BEGIN
   ZykIdx := 31;
   AntrMeld_chg_Idx := 0;
   Imp_Sek_Init := FALSE;
   OP_Mgr.Bed_aktiv := FALSE;
   OP_Mgr.Bed_ID := 0;
   OP_Mgr.Bed_Perm := 0;
   OP_Mgr.CtrlJob_act := FALSE;
   OP_Mgr.PicNum_AntrSub := FALSE;
   OP_Mgr.FM_PicNum_AntrSub := FALSE;
   OP_Mgr.PicNum_PrmSub_Rfrs := FALSE;
   OP_Mgr.PicNum_AntrSub_Rfrs := FALSE;
   OP_Mgr.MsgQuit_Zyk := FALSE;
   OP_Mgr.Bed_Perm_last := 0;
   OP_Mgr.Tmr_CtrlJob_MaxTime.ST := T#0MS;
   OP_Mgr.Tmr_CtrlJob_MaxTime.PT := T#0MS;
   OP_Mgr.Tmr_CtrlJob_MaxTime.RU := FALSE;
   OP_Mgr.Tmr_CtrlJob_MaxTime.IN := FALSE;
   OP_Mgr.Tmr_CtrlJob_BrkTime.ST := T#0MS;
   OP_Mgr.Tmr_CtrlJob_BrkTime.PT := T#0MS;
   OP_Mgr.Tmr_CtrlJob_BrkTime.RU := FALSE;
   OP_Mgr.Tmr_CtrlJob_BrkTime.IN := FALSE;
   OP_Mgr.Tmr_MsgQuit_Zyk.ST := T#0MS;
   OP_Mgr.Tmr_MsgQuit_Zyk.PT := T#0MS;
   OP_Mgr.Tmr_MsgQuit_Zyk.RU := FALSE;
   OP_Mgr.Tmr_MsgQuit_Zyk.IN := FALSE;
   OP_Mgr.CtrlJob_PicReq := 0;
   OP_Mgr.CtrlJob_PermReq := 0;
   OP_Mgr.OP_UserChg := 0;
   OP_Mgr.Antr_Idx_last := 0;
   OP_Mgr.AntrListChk_Idx := 113;
   OP_Mgr.SW_Hand_last := 0.0;
   BB_G1.Typ := 0;
   BB_G1.Idx := 0;
   BB_G1.BA_VW_Hand := FALSE;
   BB_G1.Tmr_VZ_Anlauf_Q := FALSE;
   BB_G1.SS := FALSE;
   BB_G1.SSnq := FALSE;
   BB_G1.SSfq := TRUE;
   BB_G1.nBB := FALSE;
   BB_G1.VW_Hand_St1 := FALSE;
   BB_G1.VW_Hand_St2 := FALSE;
   BB_G1.VW_Hand_Stop := FALSE;
   BB_G1.VW_Auto_St1 := FALSE;
   BB_G1.VW_Auto_St2 := FALSE;
   BB_G1.Anst_Req_St1 := FALSE;
   BB_G1.Anst_Req_St2 := FALSE;
   BB_G1.FM_Betrieb_Ein := FALSE;
   BB_G1.FM_Betrieb_Aus := TRUE;
   BB_G1.NLZ_MAZ_St1 := FALSE;
   BB_G1.NLZ_MAZ_St2 := FALSE;
   BB_G1.NLZ_Rev_SS_St1 := FALSE;
   BB_G1.NLZ_Rev_SS_St2 := FALSE;
   BB_G1.Th_St := FALSE;
   BB_G1.DMA_St := FALSE;
   BB_G1.DMZ_St := FALSE;
   BB_G1.FU_St := FALSE;
   BB_G1.TL_St := FALSE;
   BB_G1.UDr_St := FALSE;
   BB_G1.UeDr_St := FALSE;
   BB_G1.UT_St := FALSE;
   BB_G1.Le_St := FALSE;
   BB_G1.UeLM_St := FALSE;
   BB_G1.UeLE_St := FALSE;
   BB_G1.Kom_DP_St := FALSE;
   BB_G1.Kom_int_St := FALSE;
   BB_G1.int_St := FALSE;
   BB_G1.LZ_St := FALSE;
   BB_G1.BefLZ_St := FALSE;
   BB_G1.FM_GlobalQuit := FALSE;
   BB_G1.Quit_RST := FALSE;
   BB_G1.Tmr_VZ_Anlauf := 0;
   BB_G1.Tmr_VZ_ESZ := 0;
   BB_G1.Tmr_Th_St := 0;
   BB_G1.Tmr_DMA_St := 0;
   BB_G1.Tmr_DMZ_St := 0;
   BB_G1.Tmr_FU_St := 0;
   BB_G1.Tmr_TL_St := 0;
   BB_G1.Tmr_UDr_St := 0;
   BB_G1.Tmr_UeDr_St := 0;
   BB_G1.Tmr_UT_St := 0;
   BB_G1.Tmr_Le_St := 0;
   BB_G1.Tmr_UeLM_St := 0;
   BB_G1.Tmr_UeLE_St := 0;
   BB_G1.Tmr_Kom_DP_St := 0;
   BB_G1.Tmr_Kom_int_St := 0;
   BB_G1.Tmr_int_St := 0;
   BB_G1.Tmr_LZ_St := 0;
   BB_G1.Tmr_BefLZ_St := 0;
   BB_G1.Tmr_ASZ_St1 := 0;
   BB_G1.Tmr_ASZ_St2 := 0;
   BB_G1.Tmr_Rev_St1 := 0;
   BB_G1.Tmr_Rev_St2 := 0;
   BB_G1.BZ_ges_s := 507;
   BB_G1.Tmr_Quit_RST := 0;
   BB_G1.BEF_NHV.Bef.Bed_Res := FALSE;
   BB_G1.BEF_NHV.Bef.Bed_UV := FALSE;
   BB_G1.BEF_NHV.Bef.Bed_NHV := FALSE;
   BB_G1.BEF_NHV.Bef.Bed_PLS := FALSE;
   BB_G1.BEF_NHV.Bef.BA_Hand := FALSE;
   BB_G1.BEF_NHV.Bef.BA_Auto := FALSE;
   BB_G1.BEF_NHV.Bef.BF_Ein1 := FALSE;
   BB_G1.BEF_NHV.Bef.BF_Ein2 := FALSE;
   BB_G1.BEF_NHV.Bef.BF_Aus := FALSE;
   BB_G1.BEF_NHV.Bef.BZ_Res := FALSE;
   BB_G1.BEF_NHV.Bef.Res_10 := FALSE;
   BB_G1.BEF_NHV.Bef.Res_11 := FALSE;
   BB_G1.BEF_NHV.Bef.Res_12 := FALSE;
   BB_G1.BEF_NHV.Bef.Res_13 := FALSE;
   BB_G1.BEF_NHV.Bef.Res_14 := FALSE;
   BB_G1.BEF_NHV.Bef.Res_15 := FALSE;
   BB_G1.BEF_NHV.Bef.Res_16 := FALSE;
   BB_G1.BEF_NHV.Bef.Res_17 := FALSE;
   BB_G1.BEF_NHV.Bef.Res_18 := FALSE;
   BB_G1.BEF_NHV.Bef.Res_19 := FALSE;
   BB_G1.BEF_NHV.Bef.Res_20 := FALSE;
   BB_G1.BEF_NHV.Bef.Res_21 := FALSE;
   BB_G1.BEF_NHV.Bef.Res_22 := FALSE;
   BB_G1.BEF_NHV.Bef.Res_23 := FALSE;
   BB_G1.BEF_NHV.Bef.Res_24 := FALSE;
   BB_G1.BEF_NHV.Bef.Res_25 := FALSE;
   BB_G1.BEF_NHV.Bef.Res_26 := FALSE;
   BB_G1.BEF_NHV.Bef.Res_27 := FALSE;
   BB_G1.BEF_NHV.Bef.Res_28 := FALSE;
   BB_G1.BEF_NHV.Bef.Res_29 := FALSE;
   BB_G1.BEF_NHV.Bef.BF_Set_SW_chg := FALSE;
   BB_G1.BEF_NHV.Bef.BF_Quit := FALSE;
   BB_G1.BEF_NHV.SW_Hand := 0.0;
   BB_G2.Typ := 0;
   BB_G2.Idx := 1;
   BB_G2.BA_VW_Hand := FALSE;
   BB_G2.Tmr_VZ_Anlauf_Q := FALSE;
   BB_G2.SS := FALSE;
   BB_G2.SSnq := FALSE;
   BB_G2.SSfq := TRUE;
   BB_G2.nBB := FALSE;
   BB_G2.VW_Hand_St1 := FALSE;
   BB_G2.VW_Hand_St2 := FALSE;
   BB_G2.VW_Hand_Stop := FALSE;
   BB_G2.VW_Auto_St1 := FALSE;
   BB_G2.VW_Auto_St2 := FALSE;
   BB_G2.Anst_Req_St1 := FALSE;
   BB_G2.Anst_Req_St2 := FALSE;
   BB_G2.FM_Betrieb_Ein := FALSE;
   BB_G2.FM_Betrieb_Aus := TRUE;
   BB_G2.NLZ_MAZ_St1 := FALSE;
   BB_G2.NLZ_MAZ_St2 := FALSE;
   BB_G2.NLZ_Rev_SS_St1 := FALSE;
   BB_G2.NLZ_Rev_SS_St2 := FALSE;
   BB_G2.Th_St := FALSE;
   BB_G2.DMA_St := FALSE;
   BB_G2.DMZ_St := FALSE;
   BB_G2.FU_St := FALSE;
   BB_G2.TL_St := FALSE;
   BB_G2.UDr_St := FALSE;
   BB_G2.UeDr_St := FALSE;
   BB_G2.UT_St := FALSE;
   BB_G2.Le_St := FALSE;
   BB_G2.UeLM_St := FALSE;
   BB_G2.UeLE_St := FALSE;
   BB_G2.Kom_DP_St := FALSE;
   BB_G2.Kom_int_St := FALSE;
   BB_G2.int_St := FALSE;
   BB_G2.LZ_St := FALSE;
   BB_G2.BefLZ_St := FALSE;
   BB_G2.FM_GlobalQuit := FALSE;
   BB_G2.Quit_RST := FALSE;
   BB_G2.Tmr_VZ_Anlauf := 0;
   BB_G2.Tmr_VZ_ESZ := 0;
   BB_G2.Tmr_Th_St := 0;
   BB_G2.Tmr_DMA_St := 0;
   BB_G2.Tmr_DMZ_St := 0;
   BB_G2.Tmr_FU_St := 0;
   BB_G2.Tmr_TL_St := 0;
   BB_G2.Tmr_UDr_St := 0;
   BB_G2.Tmr_UeDr_St := 0;
   BB_G2.Tmr_UT_St := 0;
   BB_G2.Tmr_Le_St := 0;
   BB_G2.Tmr_UeLM_St := 0;
   BB_G2.Tmr_UeLE_St := 0;
   BB_G2.Tmr_Kom_DP_St := 0;
   BB_G2.Tmr_Kom_int_St := 0;
   BB_G2.Tmr_int_St := 0;
   BB_G2.Tmr_LZ_St := 0;
   BB_G2.Tmr_BefLZ_St := 0;
   BB_G2.Tmr_ASZ_St1 := 0;
   BB_G2.Tmr_ASZ_St2 := 0;
   BB_G2.Tmr_Rev_St1 := 0;
   BB_G2.Tmr_Rev_St2 := 0;
   BB_G2.BZ_ges_s := 3009;
   BB_G2.Tmr_Quit_RST := 0;
   BB_G2.BEF_NHV.Bef.Bed_Res := FALSE;
   BB_G2.BEF_NHV.Bef.Bed_UV := FALSE;
   BB_G2.BEF_NHV.Bef.Bed_NHV := FALSE;
   BB_G2.BEF_NHV.Bef.Bed_PLS := FALSE;
   BB_G2.BEF_NHV.Bef.BA_Hand := FALSE;
   BB_G2.BEF_NHV.Bef.BA_Auto := FALSE;
   BB_G2.BEF_NHV.Bef.BF_Ein1 := FALSE;
   BB_G2.BEF_NHV.Bef.BF_Ein2 := FALSE;
   BB_G2.BEF_NHV.Bef.BF_Aus := FALSE;
   BB_G2.BEF_NHV.Bef.BZ_Res := FALSE;
   BB_G2.BEF_NHV.Bef.Res_10 := FALSE;
   BB_G2.BEF_NHV.Bef.Res_11 := FALSE;
   BB_G2.BEF_NHV.Bef.Res_12 := FALSE;
   BB_G2.BEF_NHV.Bef.Res_13 := FALSE;
   BB_G2.BEF_NHV.Bef.Res_14 := FALSE;
   BB_G2.BEF_NHV.Bef.Res_15 := FALSE;
   BB_G2.BEF_NHV.Bef.Res_16 := FALSE;
   BB_G2.BEF_NHV.Bef.Res_17 := FALSE;
   BB_G2.BEF_NHV.Bef.Res_18 := FALSE;
   BB_G2.BEF_NHV.Bef.Res_19 := FALSE;
   BB_G2.BEF_NHV.Bef.Res_20 := FALSE;
   BB_G2.BEF_NHV.Bef.Res_21 := FALSE;
   BB_G2.BEF_NHV.Bef.Res_22 := FALSE;
   BB_G2.BEF_NHV.Bef.Res_23 := FALSE;
   BB_G2.BEF_NHV.Bef.Res_24 := FALSE;
   BB_G2.BEF_NHV.Bef.Res_25 := FALSE;
   BB_G2.BEF_NHV.Bef.Res_26 := FALSE;
   BB_G2.BEF_NHV.Bef.Res_27 := FALSE;
   BB_G2.BEF_NHV.Bef.Res_28 := FALSE;
   BB_G2.BEF_NHV.Bef.Res_29 := FALSE;
   BB_G2.BEF_NHV.Bef.BF_Set_SW_chg := FALSE;
   BB_G2.BEF_NHV.Bef.BF_Quit := FALSE;
   BB_G2.BEF_NHV.SW_Hand := 0.0;
   BB_G3.Typ := 0;
   BB_G3.Idx := 2;
   BB_G3.BA_VW_Hand := FALSE;
   BB_G3.Tmr_VZ_Anlauf_Q := FALSE;
   BB_G3.SS := FALSE;
   BB_G3.SSnq := FALSE;
   BB_G3.SSfq := TRUE;
   BB_G3.nBB := FALSE;
   BB_G3.VW_Hand_St1 := FALSE;
   BB_G3.VW_Hand_St2 := FALSE;
   BB_G3.VW_Hand_Stop := FALSE;
   BB_G3.VW_Auto_St1 := FALSE;
   BB_G3.VW_Auto_St2 := FALSE;
   BB_G3.Anst_Req_St1 := FALSE;
   BB_G3.Anst_Req_St2 := FALSE;
   BB_G3.FM_Betrieb_Ein := FALSE;
   BB_G3.FM_Betrieb_Aus := TRUE;
   BB_G3.NLZ_MAZ_St1 := FALSE;
   BB_G3.NLZ_MAZ_St2 := FALSE;
   BB_G3.NLZ_Rev_SS_St1 := FALSE;
   BB_G3.NLZ_Rev_SS_St2 := FALSE;
   BB_G3.Th_St := FALSE;
   BB_G3.DMA_St := FALSE;
   BB_G3.DMZ_St := FALSE;
   BB_G3.FU_St := FALSE;
   BB_G3.TL_St := FALSE;
   BB_G3.UDr_St := FALSE;
   BB_G3.UeDr_St := FALSE;
   BB_G3.UT_St := FALSE;
   BB_G3.Le_St := FALSE;
   BB_G3.UeLM_St := FALSE;
   BB_G3.UeLE_St := FALSE;
   BB_G3.Kom_DP_St := FALSE;
   BB_G3.Kom_int_St := FALSE;
   BB_G3.int_St := FALSE;
   BB_G3.LZ_St := FALSE;
   BB_G3.BefLZ_St := FALSE;
   BB_G3.FM_GlobalQuit := FALSE;
   BB_G3.Quit_RST := FALSE;
   BB_G3.Tmr_VZ_Anlauf := 0;
   BB_G3.Tmr_VZ_ESZ := 0;
   BB_G3.Tmr_Th_St := 0;
   BB_G3.Tmr_DMA_St := 0;
   BB_G3.Tmr_DMZ_St := 0;
   BB_G3.Tmr_FU_St := 0;
   BB_G3.Tmr_TL_St := 0;
   BB_G3.Tmr_UDr_St := 0;
   BB_G3.Tmr_UeDr_St := 0;
   BB_G3.Tmr_UT_St := 0;
   BB_G3.Tmr_Le_St := 0;
   BB_G3.Tmr_UeLM_St := 0;
   BB_G3.Tmr_UeLE_St := 0;
   BB_G3.Tmr_Kom_DP_St := 0;
   BB_G3.Tmr_Kom_int_St := 0;
   BB_G3.Tmr_int_St := 0;
   BB_G3.Tmr_LZ_St := 0;
   BB_G3.Tmr_BefLZ_St := 0;
   BB_G3.Tmr_ASZ_St1 := 0;
   BB_G3.Tmr_ASZ_St2 := 0;
   BB_G3.Tmr_Rev_St1 := 0;
   BB_G3.Tmr_Rev_St2 := 0;
   BB_G3.BZ_ges_s := 86;
   BB_G3.Tmr_Quit_RST := 0;
   BB_G3.BEF_NHV.Bef.Bed_Res := FALSE;
   BB_G3.BEF_NHV.Bef.Bed_UV := FALSE;
   BB_G3.BEF_NHV.Bef.Bed_NHV := FALSE;
   BB_G3.BEF_NHV.Bef.Bed_PLS := FALSE;
   BB_G3.BEF_NHV.Bef.BA_Hand := FALSE;
   BB_G3.BEF_NHV.Bef.BA_Auto := FALSE;
   BB_G3.BEF_NHV.Bef.BF_Ein1 := FALSE;
   BB_G3.BEF_NHV.Bef.BF_Ein2 := FALSE;
   BB_G3.BEF_NHV.Bef.BF_Aus := FALSE;
   BB_G3.BEF_NHV.Bef.BZ_Res := FALSE;
   BB_G3.BEF_NHV.Bef.Res_10 := FALSE;
   BB_G3.BEF_NHV.Bef.Res_11 := FALSE;
   BB_G3.BEF_NHV.Bef.Res_12 := FALSE;
   BB_G3.BEF_NHV.Bef.Res_13 := FALSE;
   BB_G3.BEF_NHV.Bef.Res_14 := FALSE;
   BB_G3.BEF_NHV.Bef.Res_15 := FALSE;
   BB_G3.BEF_NHV.Bef.Res_16 := FALSE;
   BB_G3.BEF_NHV.Bef.Res_17 := FALSE;
   BB_G3.BEF_NHV.Bef.Res_18 := FALSE;
   BB_G3.BEF_NHV.Bef.Res_19 := FALSE;
   BB_G3.BEF_NHV.Bef.Res_20 := FALSE;
   BB_G3.BEF_NHV.Bef.Res_21 := FALSE;
   BB_G3.BEF_NHV.Bef.Res_22 := FALSE;
   BB_G3.BEF_NHV.Bef.Res_23 := FALSE;
   BB_G3.BEF_NHV.Bef.Res_24 := FALSE;
   BB_G3.BEF_NHV.Bef.Res_25 := FALSE;
   BB_G3.BEF_NHV.Bef.Res_26 := FALSE;
   BB_G3.BEF_NHV.Bef.Res_27 := FALSE;
   BB_G3.BEF_NHV.Bef.Res_28 := FALSE;
   BB_G3.BEF_NHV.Bef.Res_29 := FALSE;
   BB_G3.BEF_NHV.Bef.BF_Set_SW_chg := FALSE;
   BB_G3.BEF_NHV.Bef.BF_Quit := FALSE;
   BB_G3.BEF_NHV.SW_Hand := 0.0;
   BB_SHL_G1.Typ := 0;
   BB_SHL_G1.Idx := 3;
   BB_SHL_G1.BA_VW_Hand := FALSE;
   BB_SHL_G1.Tmr_VZ_Anlauf_Q := FALSE;
   BB_SHL_G1.SS := FALSE;
   BB_SHL_G1.SSnq := FALSE;
   BB_SHL_G1.SSfq := TRUE;
   BB_SHL_G1.nBB := FALSE;
   BB_SHL_G1.VW_Hand_St1 := FALSE;
   BB_SHL_G1.VW_Hand_St2 := FALSE;
   BB_SHL_G1.VW_Hand_Stop := FALSE;
   BB_SHL_G1.VW_Auto_St1 := FALSE;
   BB_SHL_G1.VW_Auto_St2 := FALSE;
   BB_SHL_G1.Anst_Req_St1 := FALSE;
   BB_SHL_G1.Anst_Req_St2 := FALSE;
   BB_SHL_G1.FM_Betrieb_Ein := FALSE;
   BB_SHL_G1.FM_Betrieb_Aus := TRUE;
   BB_SHL_G1.NLZ_MAZ_St1 := FALSE;
   BB_SHL_G1.NLZ_MAZ_St2 := FALSE;
   BB_SHL_G1.NLZ_Rev_SS_St1 := FALSE;
   BB_SHL_G1.NLZ_Rev_SS_St2 := FALSE;
   BB_SHL_G1.Th_St := FALSE;
   BB_SHL_G1.DMA_St := FALSE;
   BB_SHL_G1.DMZ_St := FALSE;
   BB_SHL_G1.FU_St := FALSE;
   BB_SHL_G1.TL_St := FALSE;
   BB_SHL_G1.UDr_St := FALSE;
   BB_SHL_G1.UeDr_St := FALSE;
   BB_SHL_G1.UT_St := FALSE;
   BB_SHL_G1.Le_St := FALSE;
   BB_SHL_G1.UeLM_St := FALSE;
   BB_SHL_G1.UeLE_St := FALSE;
   BB_SHL_G1.Kom_DP_St := FALSE;
   BB_SHL_G1.Kom_int_St := FALSE;
   BB_SHL_G1.int_St := FALSE;
   BB_SHL_G1.LZ_St := FALSE;
   BB_SHL_G1.BefLZ_St := FALSE;
   BB_SHL_G1.FM_GlobalQuit := FALSE;
   BB_SHL_G1.Quit_RST := FALSE;
   BB_SHL_G1.Tmr_VZ_Anlauf := 0;
   BB_SHL_G1.Tmr_VZ_ESZ := 0;
   BB_SHL_G1.Tmr_Th_St := 0;
   BB_SHL_G1.Tmr_DMA_St := 0;
   BB_SHL_G1.Tmr_DMZ_St := 0;
   BB_SHL_G1.Tmr_FU_St := 0;
   BB_SHL_G1.Tmr_TL_St := 0;
   BB_SHL_G1.Tmr_UDr_St := 0;
   BB_SHL_G1.Tmr_UeDr_St := 0;
   BB_SHL_G1.Tmr_UT_St := 0;
   BB_SHL_G1.Tmr_Le_St := 0;
   BB_SHL_G1.Tmr_UeLM_St := 0;
   BB_SHL_G1.Tmr_UeLE_St := 0;
   BB_SHL_G1.Tmr_Kom_DP_St := 0;
   BB_SHL_G1.Tmr_Kom_int_St := 0;
   BB_SHL_G1.Tmr_int_St := 0;
   BB_SHL_G1.Tmr_LZ_St := 0;
   BB_SHL_G1.Tmr_BefLZ_St := 0;
   BB_SHL_G1.Tmr_ASZ_St1 := 0;
   BB_SHL_G1.Tmr_ASZ_St2 := 0;
   BB_SHL_G1.Tmr_Rev_St1 := 0;
   BB_SHL_G1.Tmr_Rev_St2 := 0;
   BB_SHL_G1.BZ_ges_s := 1574;
   BB_SHL_G1.Tmr_Quit_RST := 0;
   BB_SHL_G1.BEF_NHV.Bef.Bed_Res := FALSE;
   BB_SHL_G1.BEF_NHV.Bef.Bed_UV := FALSE;
   BB_SHL_G1.BEF_NHV.Bef.Bed_NHV := FALSE;
   BB_SHL_G1.BEF_NHV.Bef.Bed_PLS := FALSE;
   BB_SHL_G1.BEF_NHV.Bef.BA_Hand := FALSE;
   BB_SHL_G1.BEF_NHV.Bef.BA_Auto := FALSE;
   BB_SHL_G1.BEF_NHV.Bef.BF_Ein1 := FALSE;
   BB_SHL_G1.BEF_NHV.Bef.BF_Ein2 := FALSE;
   BB_SHL_G1.BEF_NHV.Bef.BF_Aus := FALSE;
   BB_SHL_G1.BEF_NHV.Bef.BZ_Res := FALSE;
   BB_SHL_G1.BEF_NHV.Bef.Res_10 := FALSE;
   BB_SHL_G1.BEF_NHV.Bef.Res_11 := FALSE;
   BB_SHL_G1.BEF_NHV.Bef.Res_12 := FALSE;
   BB_SHL_G1.BEF_NHV.Bef.Res_13 := FALSE;
   BB_SHL_G1.BEF_NHV.Bef.Res_14 := FALSE;
   BB_SHL_G1.BEF_NHV.Bef.Res_15 := FALSE;
   BB_SHL_G1.BEF_NHV.Bef.Res_16 := FALSE;
   BB_SHL_G1.BEF_NHV.Bef.Res_17 := FALSE;
   BB_SHL_G1.BEF_NHV.Bef.Res_18 := FALSE;
   BB_SHL_G1.BEF_NHV.Bef.Res_19 := FALSE;
   BB_SHL_G1.BEF_NHV.Bef.Res_20 := FALSE;
   BB_SHL_G1.BEF_NHV.Bef.Res_21 := FALSE;
   BB_SHL_G1.BEF_NHV.Bef.Res_22 := FALSE;
   BB_SHL_G1.BEF_NHV.Bef.Res_23 := FALSE;
   BB_SHL_G1.BEF_NHV.Bef.Res_24 := FALSE;
   BB_SHL_G1.BEF_NHV.Bef.Res_25 := FALSE;
   BB_SHL_G1.BEF_NHV.Bef.Res_26 := FALSE;
   BB_SHL_G1.BEF_NHV.Bef.Res_27 := FALSE;
   BB_SHL_G1.BEF_NHV.Bef.Res_28 := FALSE;
   BB_SHL_G1.BEF_NHV.Bef.Res_29 := FALSE;
   BB_SHL_G1.BEF_NHV.Bef.BF_Set_SW_chg := FALSE;
   BB_SHL_G1.BEF_NHV.Bef.BF_Quit := FALSE;
   BB_SHL_G1.BEF_NHV.SW_Hand := 0.0;
   BB_SHL_G2.Typ := 0;
   BB_SHL_G2.Idx := 4;
   BB_SHL_G2.BA_VW_Hand := FALSE;
   BB_SHL_G2.Tmr_VZ_Anlauf_Q := TRUE;
   BB_SHL_G2.SS := FALSE;
   BB_SHL_G2.SSnq := FALSE;
   BB_SHL_G2.SSfq := TRUE;
   BB_SHL_G2.nBB := FALSE;
   BB_SHL_G2.VW_Hand_St1 := FALSE;
   BB_SHL_G2.VW_Hand_St2 := FALSE;
   BB_SHL_G2.VW_Hand_Stop := FALSE;
   BB_SHL_G2.VW_Auto_St1 := FALSE;
   BB_SHL_G2.VW_Auto_St2 := FALSE;
   BB_SHL_G2.Anst_Req_St1 := FALSE;
   BB_SHL_G2.Anst_Req_St2 := FALSE;
   BB_SHL_G2.FM_Betrieb_Ein := TRUE;
   BB_SHL_G2.FM_Betrieb_Aus := FALSE;
   BB_SHL_G2.NLZ_MAZ_St1 := FALSE;
   BB_SHL_G2.NLZ_MAZ_St2 := FALSE;
   BB_SHL_G2.NLZ_Rev_SS_St1 := FALSE;
   BB_SHL_G2.NLZ_Rev_SS_St2 := FALSE;
   BB_SHL_G2.Th_St := FALSE;
   BB_SHL_G2.DMA_St := FALSE;
   BB_SHL_G2.DMZ_St := FALSE;
   BB_SHL_G2.FU_St := FALSE;
   BB_SHL_G2.TL_St := FALSE;
   BB_SHL_G2.UDr_St := FALSE;
   BB_SHL_G2.UeDr_St := FALSE;
   BB_SHL_G2.UT_St := FALSE;
   BB_SHL_G2.Le_St := FALSE;
   BB_SHL_G2.UeLM_St := FALSE;
   BB_SHL_G2.UeLE_St := FALSE;
   BB_SHL_G2.Kom_DP_St := FALSE;
   BB_SHL_G2.Kom_int_St := FALSE;
   BB_SHL_G2.int_St := FALSE;
   BB_SHL_G2.LZ_St := FALSE;
   BB_SHL_G2.BefLZ_St := FALSE;
   BB_SHL_G2.FM_GlobalQuit := FALSE;
   BB_SHL_G2.Quit_RST := FALSE;
   BB_SHL_G2.Tmr_VZ_Anlauf := 3;
   BB_SHL_G2.Tmr_VZ_ESZ := 0;
   BB_SHL_G2.Tmr_Th_St := 0;
   BB_SHL_G2.Tmr_DMA_St := 0;
   BB_SHL_G2.Tmr_DMZ_St := 0;
   BB_SHL_G2.Tmr_FU_St := 0;
   BB_SHL_G2.Tmr_TL_St := 0;
   BB_SHL_G2.Tmr_UDr_St := 0;
   BB_SHL_G2.Tmr_UeDr_St := 0;
   BB_SHL_G2.Tmr_UT_St := 0;
   BB_SHL_G2.Tmr_Le_St := 0;
   BB_SHL_G2.Tmr_UeLM_St := 0;
   BB_SHL_G2.Tmr_UeLE_St := 0;
   BB_SHL_G2.Tmr_Kom_DP_St := 0;
   BB_SHL_G2.Tmr_Kom_int_St := 0;
   BB_SHL_G2.Tmr_int_St := 0;
   BB_SHL_G2.Tmr_LZ_St := 0;
   BB_SHL_G2.Tmr_BefLZ_St := 0;
   BB_SHL_G2.Tmr_ASZ_St1 := 0;
   BB_SHL_G2.Tmr_ASZ_St2 := 0;
   BB_SHL_G2.Tmr_Rev_St1 := 0;
   BB_SHL_G2.Tmr_Rev_St2 := 0;
   BB_SHL_G2.BZ_ges_s := 4715;
   BB_SHL_G2.Tmr_Quit_RST := 0;
   BB_SHL_G2.BEF_NHV.Bef.Bed_Res := FALSE;
   BB_SHL_G2.BEF_NHV.Bef.Bed_UV := FALSE;
   BB_SHL_G2.BEF_NHV.Bef.Bed_NHV := FALSE;
   BB_SHL_G2.BEF_NHV.Bef.Bed_PLS := FALSE;
   BB_SHL_G2.BEF_NHV.Bef.BA_Hand := FALSE;
   BB_SHL_G2.BEF_NHV.Bef.BA_Auto := FALSE;
   BB_SHL_G2.BEF_NHV.Bef.BF_Ein1 := FALSE;
   BB_SHL_G2.BEF_NHV.Bef.BF_Ein2 := FALSE;
   BB_SHL_G2.BEF_NHV.Bef.BF_Aus := FALSE;
   BB_SHL_G2.BEF_NHV.Bef.BZ_Res := FALSE;
   BB_SHL_G2.BEF_NHV.Bef.Res_10 := FALSE;
   BB_SHL_G2.BEF_NHV.Bef.Res_11 := FALSE;
   BB_SHL_G2.BEF_NHV.Bef.Res_12 := FALSE;
   BB_SHL_G2.BEF_NHV.Bef.Res_13 := FALSE;
   BB_SHL_G2.BEF_NHV.Bef.Res_14 := FALSE;
   BB_SHL_G2.BEF_NHV.Bef.Res_15 := FALSE;
   BB_SHL_G2.BEF_NHV.Bef.Res_16 := FALSE;
   BB_SHL_G2.BEF_NHV.Bef.Res_17 := FALSE;
   BB_SHL_G2.BEF_NHV.Bef.Res_18 := FALSE;
   BB_SHL_G2.BEF_NHV.Bef.Res_19 := FALSE;
   BB_SHL_G2.BEF_NHV.Bef.Res_20 := FALSE;
   BB_SHL_G2.BEF_NHV.Bef.Res_21 := FALSE;
   BB_SHL_G2.BEF_NHV.Bef.Res_22 := FALSE;
   BB_SHL_G2.BEF_NHV.Bef.Res_23 := FALSE;
   BB_SHL_G2.BEF_NHV.Bef.Res_24 := FALSE;
   BB_SHL_G2.BEF_NHV.Bef.Res_25 := FALSE;
   BB_SHL_G2.BEF_NHV.Bef.Res_26 := FALSE;
   BB_SHL_G2.BEF_NHV.Bef.Res_27 := FALSE;
   BB_SHL_G2.BEF_NHV.Bef.Res_28 := FALSE;
   BB_SHL_G2.BEF_NHV.Bef.Res_29 := FALSE;
   BB_SHL_G2.BEF_NHV.Bef.BF_Set_SW_chg := FALSE;
   BB_SHL_G2.BEF_NHV.Bef.BF_Quit := FALSE;
   BB_SHL_G2.BEF_NHV.SW_Hand := 0.0;
   BB_SHL_G3.Typ := 0;
   BB_SHL_G3.Idx := 5;
   BB_SHL_G3.BA_VW_Hand := FALSE;
   BB_SHL_G3.Tmr_VZ_Anlauf_Q := FALSE;
   BB_SHL_G3.SS := FALSE;
   BB_SHL_G3.SSnq := FALSE;
   BB_SHL_G3.SSfq := TRUE;
   BB_SHL_G3.nBB := FALSE;
   BB_SHL_G3.VW_Hand_St1 := FALSE;
   BB_SHL_G3.VW_Hand_St2 := FALSE;
   BB_SHL_G3.VW_Hand_Stop := FALSE;
   BB_SHL_G3.VW_Auto_St1 := FALSE;
   BB_SHL_G3.VW_Auto_St2 := FALSE;
   BB_SHL_G3.Anst_Req_St1 := FALSE;
   BB_SHL_G3.Anst_Req_St2 := FALSE;
   BB_SHL_G3.FM_Betrieb_Ein := FALSE;
   BB_SHL_G3.FM_Betrieb_Aus := TRUE;
   BB_SHL_G3.NLZ_MAZ_St1 := FALSE;
   BB_SHL_G3.NLZ_MAZ_St2 := FALSE;
   BB_SHL_G3.NLZ_Rev_SS_St1 := FALSE;
   BB_SHL_G3.NLZ_Rev_SS_St2 := FALSE;
   BB_SHL_G3.Th_St := FALSE;
   BB_SHL_G3.DMA_St := FALSE;
   BB_SHL_G3.DMZ_St := FALSE;
   BB_SHL_G3.FU_St := FALSE;
   BB_SHL_G3.TL_St := FALSE;
   BB_SHL_G3.UDr_St := FALSE;
   BB_SHL_G3.UeDr_St := FALSE;
   BB_SHL_G3.UT_St := FALSE;
   BB_SHL_G3.Le_St := FALSE;
   BB_SHL_G3.UeLM_St := FALSE;
   BB_SHL_G3.UeLE_St := FALSE;
   BB_SHL_G3.Kom_DP_St := FALSE;
   BB_SHL_G3.Kom_int_St := FALSE;
   BB_SHL_G3.int_St := FALSE;
   BB_SHL_G3.LZ_St := FALSE;
   BB_SHL_G3.BefLZ_St := FALSE;
   BB_SHL_G3.FM_GlobalQuit := FALSE;
   BB_SHL_G3.Quit_RST := FALSE;
   BB_SHL_G3.Tmr_VZ_Anlauf := 0;
   BB_SHL_G3.Tmr_VZ_ESZ := 0;
   BB_SHL_G3.Tmr_Th_St := 0;
   BB_SHL_G3.Tmr_DMA_St := 0;
   BB_SHL_G3.Tmr_DMZ_St := 0;
   BB_SHL_G3.Tmr_FU_St := 0;
   BB_SHL_G3.Tmr_TL_St := 0;
   BB_SHL_G3.Tmr_UDr_St := 0;
   BB_SHL_G3.Tmr_UeDr_St := 0;
   BB_SHL_G3.Tmr_UT_St := 0;
   BB_SHL_G3.Tmr_Le_St := 0;
   BB_SHL_G3.Tmr_UeLM_St := 0;
   BB_SHL_G3.Tmr_UeLE_St := 0;
   BB_SHL_G3.Tmr_Kom_DP_St := 0;
   BB_SHL_G3.Tmr_Kom_int_St := 0;
   BB_SHL_G3.Tmr_int_St := 0;
   BB_SHL_G3.Tmr_LZ_St := 0;
   BB_SHL_G3.Tmr_BefLZ_St := 0;
   BB_SHL_G3.Tmr_ASZ_St1 := 0;
   BB_SHL_G3.Tmr_ASZ_St2 := 0;
   BB_SHL_G3.Tmr_Rev_St1 := 0;
   BB_SHL_G3.Tmr_Rev_St2 := 0;
   BB_SHL_G3.BZ_ges_s := 1375;
   BB_SHL_G3.Tmr_Quit_RST := 0;
   BB_SHL_G3.BEF_NHV.Bef.Bed_Res := FALSE;
   BB_SHL_G3.BEF_NHV.Bef.Bed_UV := FALSE;
   BB_SHL_G3.BEF_NHV.Bef.Bed_NHV := FALSE;
   BB_SHL_G3.BEF_NHV.Bef.Bed_PLS := FALSE;
   BB_SHL_G3.BEF_NHV.Bef.BA_Hand := FALSE;
   BB_SHL_G3.BEF_NHV.Bef.BA_Auto := FALSE;
   BB_SHL_G3.BEF_NHV.Bef.BF_Ein1 := FALSE;
   BB_SHL_G3.BEF_NHV.Bef.BF_Ein2 := FALSE;
   BB_SHL_G3.BEF_NHV.Bef.BF_Aus := FALSE;
   BB_SHL_G3.BEF_NHV.Bef.BZ_Res := FALSE;
   BB_SHL_G3.BEF_NHV.Bef.Res_10 := FALSE;
   BB_SHL_G3.BEF_NHV.Bef.Res_11 := FALSE;
   BB_SHL_G3.BEF_NHV.Bef.Res_12 := FALSE;
   BB_SHL_G3.BEF_NHV.Bef.Res_13 := FALSE;
   BB_SHL_G3.BEF_NHV.Bef.Res_14 := FALSE;
   BB_SHL_G3.BEF_NHV.Bef.Res_15 := FALSE;
   BB_SHL_G3.BEF_NHV.Bef.Res_16 := FALSE;
   BB_SHL_G3.BEF_NHV.Bef.Res_17 := FALSE;
   BB_SHL_G3.BEF_NHV.Bef.Res_18 := FALSE;
   BB_SHL_G3.BEF_NHV.Bef.Res_19 := FALSE;
   BB_SHL_G3.BEF_NHV.Bef.Res_20 := FALSE;
   BB_SHL_G3.BEF_NHV.Bef.Res_21 := FALSE;
   BB_SHL_G3.BEF_NHV.Bef.Res_22 := FALSE;
   BB_SHL_G3.BEF_NHV.Bef.Res_23 := FALSE;
   BB_SHL_G3.BEF_NHV.Bef.Res_24 := FALSE;
   BB_SHL_G3.BEF_NHV.Bef.Res_25 := FALSE;
   BB_SHL_G3.BEF_NHV.Bef.Res_26 := FALSE;
   BB_SHL_G3.BEF_NHV.Bef.Res_27 := FALSE;
   BB_SHL_G3.BEF_NHV.Bef.Res_28 := FALSE;
   BB_SHL_G3.BEF_NHV.Bef.Res_29 := FALSE;
   BB_SHL_G3.BEF_NHV.Bef.BF_Set_SW_chg := FALSE;
   BB_SHL_G3.BEF_NHV.Bef.BF_Quit := FALSE;
   BB_SHL_G3.BEF_NHV.SW_Hand := 0.0;
   BB_AV.Typ := 0;
   BB_AV.Idx := 6;
   BB_AV.BA_VW_Hand := FALSE;
   BB_AV.Tmr_VZ_Anlauf_Q := FALSE;
   BB_AV.SS := FALSE;
   BB_AV.SSnq := FALSE;
   BB_AV.SSfq := TRUE;
   BB_AV.nBB := FALSE;
   BB_AV.VW_Hand_St1 := FALSE;
   BB_AV.VW_Hand_St2 := FALSE;
   BB_AV.VW_Hand_Stop := FALSE;
   BB_AV.VW_Auto_St1 := FALSE;
   BB_AV.VW_Auto_St2 := FALSE;
   BB_AV.Anst_Req_St1 := FALSE;
   BB_AV.Anst_Req_St2 := FALSE;
   BB_AV.FM_Betrieb_Ein := FALSE;
   BB_AV.FM_Betrieb_Aus := TRUE;
   BB_AV.NLZ_MAZ_St1 := FALSE;
   BB_AV.NLZ_MAZ_St2 := FALSE;
   BB_AV.NLZ_Rev_SS_St1 := FALSE;
   BB_AV.NLZ_Rev_SS_St2 := FALSE;
   BB_AV.Th_St := FALSE;
   BB_AV.DMA_St := FALSE;
   BB_AV.DMZ_St := FALSE;
   BB_AV.FU_St := FALSE;
   BB_AV.TL_St := FALSE;
   BB_AV.UDr_St := FALSE;
   BB_AV.UeDr_St := FALSE;
   BB_AV.UT_St := FALSE;
   BB_AV.Le_St := FALSE;
   BB_AV.UeLM_St := FALSE;
   BB_AV.UeLE_St := FALSE;
   BB_AV.Kom_DP_St := FALSE;
   BB_AV.Kom_int_St := FALSE;
   BB_AV.int_St := FALSE;
   BB_AV.LZ_St := FALSE;
   BB_AV.BefLZ_St := FALSE;
   BB_AV.FM_GlobalQuit := FALSE;
   BB_AV.Quit_RST := FALSE;
   BB_AV.Tmr_VZ_Anlauf := 0;
   BB_AV.Tmr_VZ_ESZ := 0;
   BB_AV.Tmr_Th_St := 0;
   BB_AV.Tmr_DMA_St := 0;
   BB_AV.Tmr_DMZ_St := 0;
   BB_AV.Tmr_FU_St := 0;
   BB_AV.Tmr_TL_St := 0;
   BB_AV.Tmr_UDr_St := 0;
   BB_AV.Tmr_UeDr_St := 0;
   BB_AV.Tmr_UT_St := 0;
   BB_AV.Tmr_Le_St := 0;
   BB_AV.Tmr_UeLM_St := 0;
   BB_AV.Tmr_UeLE_St := 0;
   BB_AV.Tmr_Kom_DP_St := 0;
   BB_AV.Tmr_Kom_int_St := 0;
   BB_AV.Tmr_int_St := 0;
   BB_AV.Tmr_LZ_St := 0;
   BB_AV.Tmr_BefLZ_St := 0;
   BB_AV.Tmr_ASZ_St1 := 0;
   BB_AV.Tmr_ASZ_St2 := 0;
   BB_AV.Tmr_Rev_St1 := 0;
   BB_AV.Tmr_Rev_St2 := 0;
   BB_AV.BZ_ges_s := 0;
   BB_AV.Tmr_Quit_RST := 0;
   BB_AV.BEF_NHV.Bef.Bed_Res := FALSE;
   BB_AV.BEF_NHV.Bef.Bed_UV := FALSE;
   BB_AV.BEF_NHV.Bef.Bed_NHV := FALSE;
   BB_AV.BEF_NHV.Bef.Bed_PLS := FALSE;
   BB_AV.BEF_NHV.Bef.BA_Hand := FALSE;
   BB_AV.BEF_NHV.Bef.BA_Auto := FALSE;
   BB_AV.BEF_NHV.Bef.BF_Ein1 := FALSE;
   BB_AV.BEF_NHV.Bef.BF_Ein2 := FALSE;
   BB_AV.BEF_NHV.Bef.BF_Aus := FALSE;
   BB_AV.BEF_NHV.Bef.BZ_Res := FALSE;
   BB_AV.BEF_NHV.Bef.Res_10 := FALSE;
   BB_AV.BEF_NHV.Bef.Res_11 := FALSE;
   BB_AV.BEF_NHV.Bef.Res_12 := FALSE;
   BB_AV.BEF_NHV.Bef.Res_13 := FALSE;
   BB_AV.BEF_NHV.Bef.Res_14 := FALSE;
   BB_AV.BEF_NHV.Bef.Res_15 := FALSE;
   BB_AV.BEF_NHV.Bef.Res_16 := FALSE;
   BB_AV.BEF_NHV.Bef.Res_17 := FALSE;
   BB_AV.BEF_NHV.Bef.Res_18 := FALSE;
   BB_AV.BEF_NHV.Bef.Res_19 := FALSE;
   BB_AV.BEF_NHV.Bef.Res_20 := FALSE;
   BB_AV.BEF_NHV.Bef.Res_21 := FALSE;
   BB_AV.BEF_NHV.Bef.Res_22 := FALSE;
   BB_AV.BEF_NHV.Bef.Res_23 := FALSE;
   BB_AV.BEF_NHV.Bef.Res_24 := FALSE;
   BB_AV.BEF_NHV.Bef.Res_25 := FALSE;
   BB_AV.BEF_NHV.Bef.Res_26 := FALSE;
   BB_AV.BEF_NHV.Bef.Res_27 := FALSE;
   BB_AV.BEF_NHV.Bef.Res_28 := FALSE;
   BB_AV.BEF_NHV.Bef.Res_29 := FALSE;
   BB_AV.BEF_NHV.Bef.BF_Set_SW_chg := FALSE;
   BB_AV.BEF_NHV.Bef.BF_Quit := FALSE;
   BB_AV.BEF_NHV.SW_Hand := 0.0;
   BB_LS1.Typ := 5;
   BB_LS1.Idx := 7;
   BB_LS1.BA_VW_Hand := FALSE;
   BB_LS1.Tmr_VZ_Anlauf_Q := FALSE;
   BB_LS1.SS := FALSE;
   BB_LS1.SSnq := FALSE;
   BB_LS1.SSfq := TRUE;
   BB_LS1.nBB := FALSE;
   BB_LS1.VW_Hand_St1 := FALSE;
   BB_LS1.VW_Hand_St2 := FALSE;
   BB_LS1.VW_Hand_Stop := FALSE;
   BB_LS1.VW_Auto_St1 := FALSE;
   BB_LS1.VW_Auto_St2 := FALSE;
   BB_LS1.Anst_Req_St1 := FALSE;
   BB_LS1.Anst_Req_St2 := FALSE;
   BB_LS1.FM_Betrieb_Ein := FALSE;
   BB_LS1.FM_Betrieb_Aus := TRUE;
   BB_LS1.NLZ_MAZ_St1 := FALSE;
   BB_LS1.NLZ_MAZ_St2 := FALSE;
   BB_LS1.NLZ_Rev_SS_St1 := FALSE;
   BB_LS1.NLZ_Rev_SS_St2 := FALSE;
   BB_LS1.Th_St := FALSE;
   BB_LS1.DMA_St := FALSE;
   BB_LS1.DMZ_St := FALSE;
   BB_LS1.FU_St := FALSE;
   BB_LS1.TL_St := FALSE;
   BB_LS1.UDr_St := FALSE;
   BB_LS1.UeDr_St := FALSE;
   BB_LS1.UT_St := FALSE;
   BB_LS1.Le_St := FALSE;
   BB_LS1.UeLM_St := FALSE;
   BB_LS1.UeLE_St := FALSE;
   BB_LS1.Kom_DP_St := FALSE;
   BB_LS1.Kom_int_St := FALSE;
   BB_LS1.int_St := FALSE;
   BB_LS1.LZ_St := FALSE;
   BB_LS1.BefLZ_St := FALSE;
   BB_LS1.FM_GlobalQuit := FALSE;
   BB_LS1.Quit_RST := FALSE;
   BB_LS1.Tmr_VZ_Anlauf := 0;
   BB_LS1.Tmr_VZ_ESZ := 0;
   BB_LS1.Tmr_Th_St := 0;
   BB_LS1.Tmr_DMA_St := 0;
   BB_LS1.Tmr_DMZ_St := 0;
   BB_LS1.Tmr_FU_St := 0;
   BB_LS1.Tmr_TL_St := 0;
   BB_LS1.Tmr_UDr_St := 0;
   BB_LS1.Tmr_UeDr_St := 0;
   BB_LS1.Tmr_UT_St := 0;
   BB_LS1.Tmr_Le_St := 0;
   BB_LS1.Tmr_UeLM_St := 0;
   BB_LS1.Tmr_UeLE_St := 0;
   BB_LS1.Tmr_Kom_DP_St := 0;
   BB_LS1.Tmr_Kom_int_St := 0;
   BB_LS1.Tmr_int_St := 0;
   BB_LS1.Tmr_LZ_St := 0;
   BB_LS1.Tmr_BefLZ_St := 0;
   BB_LS1.Tmr_ASZ_St1 := 0;
   BB_LS1.Tmr_ASZ_St2 := 0;
   BB_LS1.Tmr_Rev_St1 := 0;
   BB_LS1.Tmr_Rev_St2 := 0;
   BB_LS1.BZ_ges_s := 127;
   BB_LS1.Tmr_Quit_RST := 0;
   BB_LS1.BEF_NHV.Bef.Bed_Res := FALSE;
   BB_LS1.BEF_NHV.Bef.Bed_UV := FALSE;
   BB_LS1.BEF_NHV.Bef.Bed_NHV := FALSE;
   BB_LS1.BEF_NHV.Bef.Bed_PLS := FALSE;
   BB_LS1.BEF_NHV.Bef.BA_Hand := FALSE;
   BB_LS1.BEF_NHV.Bef.BA_Auto := FALSE;
   BB_LS1.BEF_NHV.Bef.BF_Ein1 := FALSE;
   BB_LS1.BEF_NHV.Bef.BF_Ein2 := FALSE;
   BB_LS1.BEF_NHV.Bef.BF_Aus := FALSE;
   BB_LS1.BEF_NHV.Bef.BZ_Res := FALSE;
   BB_LS1.BEF_NHV.Bef.Res_10 := FALSE;
   BB_LS1.BEF_NHV.Bef.Res_11 := FALSE;
   BB_LS1.BEF_NHV.Bef.Res_12 := FALSE;
   BB_LS1.BEF_NHV.Bef.Res_13 := FALSE;
   BB_LS1.BEF_NHV.Bef.Res_14 := FALSE;
   BB_LS1.BEF_NHV.Bef.Res_15 := FALSE;
   BB_LS1.BEF_NHV.Bef.Res_16 := FALSE;
   BB_LS1.BEF_NHV.Bef.Res_17 := FALSE;
   BB_LS1.BEF_NHV.Bef.Res_18 := FALSE;
   BB_LS1.BEF_NHV.Bef.Res_19 := FALSE;
   BB_LS1.BEF_NHV.Bef.Res_20 := FALSE;
   BB_LS1.BEF_NHV.Bef.Res_21 := FALSE;
   BB_LS1.BEF_NHV.Bef.Res_22 := FALSE;
   BB_LS1.BEF_NHV.Bef.Res_23 := FALSE;
   BB_LS1.BEF_NHV.Bef.Res_24 := FALSE;
   BB_LS1.BEF_NHV.Bef.Res_25 := FALSE;
   BB_LS1.BEF_NHV.Bef.Res_26 := FALSE;
   BB_LS1.BEF_NHV.Bef.Res_27 := FALSE;
   BB_LS1.BEF_NHV.Bef.Res_28 := FALSE;
   BB_LS1.BEF_NHV.Bef.Res_29 := FALSE;
   BB_LS1.BEF_NHV.Bef.BF_Set_SW_chg := FALSE;
   BB_LS1.BEF_NHV.Bef.BF_Quit := FALSE;
   BB_LS1.BEF_NHV.SW_Hand := 0.0;
   BB_LS2.Typ := 5;
   BB_LS2.Idx := 8;
   BB_LS2.BA_VW_Hand := FALSE;
   BB_LS2.Tmr_VZ_Anlauf_Q := FALSE;
   BB_LS2.SS := FALSE;
   BB_LS2.SSnq := FALSE;
   BB_LS2.SSfq := TRUE;
   BB_LS2.nBB := FALSE;
   BB_LS2.VW_Hand_St1 := FALSE;
   BB_LS2.VW_Hand_St2 := FALSE;
   BB_LS2.VW_Hand_Stop := FALSE;
   BB_LS2.VW_Auto_St1 := FALSE;
   BB_LS2.VW_Auto_St2 := FALSE;
   BB_LS2.Anst_Req_St1 := FALSE;
   BB_LS2.Anst_Req_St2 := FALSE;
   BB_LS2.FM_Betrieb_Ein := FALSE;
   BB_LS2.FM_Betrieb_Aus := TRUE;
   BB_LS2.NLZ_MAZ_St1 := FALSE;
   BB_LS2.NLZ_MAZ_St2 := FALSE;
   BB_LS2.NLZ_Rev_SS_St1 := FALSE;
   BB_LS2.NLZ_Rev_SS_St2 := FALSE;
   BB_LS2.Th_St := FALSE;
   BB_LS2.DMA_St := FALSE;
   BB_LS2.DMZ_St := FALSE;
   BB_LS2.FU_St := FALSE;
   BB_LS2.TL_St := FALSE;
   BB_LS2.UDr_St := FALSE;
   BB_LS2.UeDr_St := FALSE;
   BB_LS2.UT_St := FALSE;
   BB_LS2.Le_St := FALSE;
   BB_LS2.UeLM_St := FALSE;
   BB_LS2.UeLE_St := FALSE;
   BB_LS2.Kom_DP_St := FALSE;
   BB_LS2.Kom_int_St := FALSE;
   BB_LS2.int_St := FALSE;
   BB_LS2.LZ_St := FALSE;
   BB_LS2.BefLZ_St := FALSE;
   BB_LS2.FM_GlobalQuit := FALSE;
   BB_LS2.Quit_RST := FALSE;
   BB_LS2.Tmr_VZ_Anlauf := 0;
   BB_LS2.Tmr_VZ_ESZ := 0;
   BB_LS2.Tmr_Th_St := 0;
   BB_LS2.Tmr_DMA_St := 0;
   BB_LS2.Tmr_DMZ_St := 0;
   BB_LS2.Tmr_FU_St := 0;
   BB_LS2.Tmr_TL_St := 0;
   BB_LS2.Tmr_UDr_St := 0;
   BB_LS2.Tmr_UeDr_St := 0;
   BB_LS2.Tmr_UT_St := 0;
   BB_LS2.Tmr_Le_St := 0;
   BB_LS2.Tmr_UeLM_St := 0;
   BB_LS2.Tmr_UeLE_St := 0;
   BB_LS2.Tmr_Kom_DP_St := 0;
   BB_LS2.Tmr_Kom_int_St := 0;
   BB_LS2.Tmr_int_St := 0;
   BB_LS2.Tmr_LZ_St := 0;
   BB_LS2.Tmr_BefLZ_St := 0;
   BB_LS2.Tmr_ASZ_St1 := 0;
   BB_LS2.Tmr_ASZ_St2 := 0;
   BB_LS2.Tmr_Rev_St1 := 0;
   BB_LS2.Tmr_Rev_St2 := 0;
   BB_LS2.BZ_ges_s := 298;
   BB_LS2.Tmr_Quit_RST := 0;
   BB_LS2.BEF_NHV.Bef.Bed_Res := FALSE;
   BB_LS2.BEF_NHV.Bef.Bed_UV := FALSE;
   BB_LS2.BEF_NHV.Bef.Bed_NHV := FALSE;
   BB_LS2.BEF_NHV.Bef.Bed_PLS := FALSE;
   BB_LS2.BEF_NHV.Bef.BA_Hand := FALSE;
   BB_LS2.BEF_NHV.Bef.BA_Auto := FALSE;
   BB_LS2.BEF_NHV.Bef.BF_Ein1 := FALSE;
   BB_LS2.BEF_NHV.Bef.BF_Ein2 := FALSE;
   BB_LS2.BEF_NHV.Bef.BF_Aus := FALSE;
   BB_LS2.BEF_NHV.Bef.BZ_Res := FALSE;
   BB_LS2.BEF_NHV.Bef.Res_10 := FALSE;
   BB_LS2.BEF_NHV.Bef.Res_11 := FALSE;
   BB_LS2.BEF_NHV.Bef.Res_12 := FALSE;
   BB_LS2.BEF_NHV.Bef.Res_13 := FALSE;
   BB_LS2.BEF_NHV.Bef.Res_14 := FALSE;
   BB_LS2.BEF_NHV.Bef.Res_15 := FALSE;
   BB_LS2.BEF_NHV.Bef.Res_16 := FALSE;
   BB_LS2.BEF_NHV.Bef.Res_17 := FALSE;
   BB_LS2.BEF_NHV.Bef.Res_18 := FALSE;
   BB_LS2.BEF_NHV.Bef.Res_19 := FALSE;
   BB_LS2.BEF_NHV.Bef.Res_20 := FALSE;
   BB_LS2.BEF_NHV.Bef.Res_21 := FALSE;
   BB_LS2.BEF_NHV.Bef.Res_22 := FALSE;
   BB_LS2.BEF_NHV.Bef.Res_23 := FALSE;
   BB_LS2.BEF_NHV.Bef.Res_24 := FALSE;
   BB_LS2.BEF_NHV.Bef.Res_25 := FALSE;
   BB_LS2.BEF_NHV.Bef.Res_26 := FALSE;
   BB_LS2.BEF_NHV.Bef.Res_27 := FALSE;
   BB_LS2.BEF_NHV.Bef.Res_28 := FALSE;
   BB_LS2.BEF_NHV.Bef.Res_29 := FALSE;
   BB_LS2.BEF_NHV.Bef.BF_Set_SW_chg := FALSE;
   BB_LS2.BEF_NHV.Bef.BF_Quit := FALSE;
   BB_LS2.BEF_NHV.SW_Hand := 0.0;
   BB1_RZP1.Typ := 0;
   BB1_RZP1.Idx := 9;
   BB1_RZP1.BA_VW_Hand := FALSE;
   BB1_RZP1.Tmr_VZ_Anlauf_Q := TRUE;
   BB1_RZP1.SS := FALSE;
   BB1_RZP1.SSnq := FALSE;
   BB1_RZP1.SSfq := TRUE;
   BB1_RZP1.nBB := FALSE;
   BB1_RZP1.VW_Hand_St1 := FALSE;
   BB1_RZP1.VW_Hand_St2 := FALSE;
   BB1_RZP1.VW_Hand_Stop := FALSE;
   BB1_RZP1.VW_Auto_St1 := TRUE;
   BB1_RZP1.VW_Auto_St2 := FALSE;
   BB1_RZP1.Anst_Req_St1 := TRUE;
   BB1_RZP1.Anst_Req_St2 := FALSE;
   BB1_RZP1.FM_Betrieb_Ein := TRUE;
   BB1_RZP1.FM_Betrieb_Aus := FALSE;
   BB1_RZP1.NLZ_MAZ_St1 := TRUE;
   BB1_RZP1.NLZ_MAZ_St2 := FALSE;
   BB1_RZP1.NLZ_Rev_SS_St1 := TRUE;
   BB1_RZP1.NLZ_Rev_SS_St2 := FALSE;
   BB1_RZP1.Th_St := FALSE;
   BB1_RZP1.DMA_St := FALSE;
   BB1_RZP1.DMZ_St := FALSE;
   BB1_RZP1.FU_St := FALSE;
   BB1_RZP1.TL_St := FALSE;
   BB1_RZP1.UDr_St := FALSE;
   BB1_RZP1.UeDr_St := FALSE;
   BB1_RZP1.UT_St := FALSE;
   BB1_RZP1.Le_St := FALSE;
   BB1_RZP1.UeLM_St := FALSE;
   BB1_RZP1.UeLE_St := FALSE;
   BB1_RZP1.Kom_DP_St := FALSE;
   BB1_RZP1.Kom_int_St := FALSE;
   BB1_RZP1.int_St := FALSE;
   BB1_RZP1.LZ_St := FALSE;
   BB1_RZP1.BefLZ_St := FALSE;
   BB1_RZP1.FM_GlobalQuit := FALSE;
   BB1_RZP1.Quit_RST := FALSE;
   BB1_RZP1.Tmr_VZ_Anlauf := 3;
   BB1_RZP1.Tmr_VZ_ESZ := 0;
   BB1_RZP1.Tmr_Th_St := 0;
   BB1_RZP1.Tmr_DMA_St := 0;
   BB1_RZP1.Tmr_DMZ_St := 0;
   BB1_RZP1.Tmr_FU_St := 0;
   BB1_RZP1.Tmr_TL_St := 0;
   BB1_RZP1.Tmr_UDr_St := 0;
   BB1_RZP1.Tmr_UeDr_St := 0;
   BB1_RZP1.Tmr_UT_St := 0;
   BB1_RZP1.Tmr_Le_St := 0;
   BB1_RZP1.Tmr_UeLM_St := 0;
   BB1_RZP1.Tmr_UeLE_St := 0;
   BB1_RZP1.Tmr_Kom_DP_St := 0;
   BB1_RZP1.Tmr_Kom_int_St := 0;
   BB1_RZP1.Tmr_int_St := 0;
   BB1_RZP1.Tmr_LZ_St := 0;
   BB1_RZP1.Tmr_BefLZ_St := 0;
   BB1_RZP1.Tmr_ASZ_St1 := 5;
   BB1_RZP1.Tmr_ASZ_St2 := 0;
   BB1_RZP1.Tmr_Rev_St1 := 10;
   BB1_RZP1.Tmr_Rev_St2 := 0;
   BB1_RZP1.BZ_ges_s := 2190;
   BB1_RZP1.Tmr_Quit_RST := 0;
   BB1_RZP1.BEF_NHV.Bef.Bed_Res := FALSE;
   BB1_RZP1.BEF_NHV.Bef.Bed_UV := FALSE;
   BB1_RZP1.BEF_NHV.Bef.Bed_NHV := FALSE;
   BB1_RZP1.BEF_NHV.Bef.Bed_PLS := FALSE;
   BB1_RZP1.BEF_NHV.Bef.BA_Hand := FALSE;
   BB1_RZP1.BEF_NHV.Bef.BA_Auto := FALSE;
   BB1_RZP1.BEF_NHV.Bef.BF_Ein1 := FALSE;
   BB1_RZP1.BEF_NHV.Bef.BF_Ein2 := FALSE;
   BB1_RZP1.BEF_NHV.Bef.BF_Aus := FALSE;
   BB1_RZP1.BEF_NHV.Bef.BZ_Res := FALSE;
   BB1_RZP1.BEF_NHV.Bef.Res_10 := FALSE;
   BB1_RZP1.BEF_NHV.Bef.Res_11 := FALSE;
   BB1_RZP1.BEF_NHV.Bef.Res_12 := FALSE;
   BB1_RZP1.BEF_NHV.Bef.Res_13 := FALSE;
   BB1_RZP1.BEF_NHV.Bef.Res_14 := FALSE;
   BB1_RZP1.BEF_NHV.Bef.Res_15 := FALSE;
   BB1_RZP1.BEF_NHV.Bef.Res_16 := FALSE;
   BB1_RZP1.BEF_NHV.Bef.Res_17 := FALSE;
   BB1_RZP1.BEF_NHV.Bef.Res_18 := FALSE;
   BB1_RZP1.BEF_NHV.Bef.Res_19 := FALSE;
   BB1_RZP1.BEF_NHV.Bef.Res_20 := FALSE;
   BB1_RZP1.BEF_NHV.Bef.Res_21 := FALSE;
   BB1_RZP1.BEF_NHV.Bef.Res_22 := FALSE;
   BB1_RZP1.BEF_NHV.Bef.Res_23 := FALSE;
   BB1_RZP1.BEF_NHV.Bef.Res_24 := FALSE;
   BB1_RZP1.BEF_NHV.Bef.Res_25 := FALSE;
   BB1_RZP1.BEF_NHV.Bef.Res_26 := FALSE;
   BB1_RZP1.BEF_NHV.Bef.Res_27 := FALSE;
   BB1_RZP1.BEF_NHV.Bef.Res_28 := FALSE;
   BB1_RZP1.BEF_NHV.Bef.Res_29 := FALSE;
   BB1_RZP1.BEF_NHV.Bef.BF_Set_SW_chg := FALSE;
   BB1_RZP1.BEF_NHV.Bef.BF_Quit := FALSE;
   BB1_RZP1.BEF_NHV.SW_Hand := 0.0;
   BB1_RZP2.Typ := 0;
   BB1_RZP2.Idx := 10;
   BB1_RZP2.BA_VW_Hand := FALSE;
   BB1_RZP2.Tmr_VZ_Anlauf_Q := FALSE;
   BB1_RZP2.SS := FALSE;
   BB1_RZP2.SSnq := FALSE;
   BB1_RZP2.SSfq := TRUE;
   BB1_RZP2.nBB := FALSE;
   BB1_RZP2.VW_Hand_St1 := FALSE;
   BB1_RZP2.VW_Hand_St2 := FALSE;
   BB1_RZP2.VW_Hand_Stop := FALSE;
   BB1_RZP2.VW_Auto_St1 := FALSE;
   BB1_RZP2.VW_Auto_St2 := FALSE;
   BB1_RZP2.Anst_Req_St1 := FALSE;
   BB1_RZP2.Anst_Req_St2 := FALSE;
   BB1_RZP2.FM_Betrieb_Ein := FALSE;
   BB1_RZP2.FM_Betrieb_Aus := TRUE;
   BB1_RZP2.NLZ_MAZ_St1 := FALSE;
   BB1_RZP2.NLZ_MAZ_St2 := FALSE;
   BB1_RZP2.NLZ_Rev_SS_St1 := FALSE;
   BB1_RZP2.NLZ_Rev_SS_St2 := FALSE;
   BB1_RZP2.Th_St := FALSE;
   BB1_RZP2.DMA_St := FALSE;
   BB1_RZP2.DMZ_St := FALSE;
   BB1_RZP2.FU_St := FALSE;
   BB1_RZP2.TL_St := FALSE;
   BB1_RZP2.UDr_St := FALSE;
   BB1_RZP2.UeDr_St := FALSE;
   BB1_RZP2.UT_St := FALSE;
   BB1_RZP2.Le_St := FALSE;
   BB1_RZP2.UeLM_St := FALSE;
   BB1_RZP2.UeLE_St := FALSE;
   BB1_RZP2.Kom_DP_St := FALSE;
   BB1_RZP2.Kom_int_St := FALSE;
   BB1_RZP2.int_St := FALSE;
   BB1_RZP2.LZ_St := FALSE;
   BB1_RZP2.BefLZ_St := FALSE;
   BB1_RZP2.FM_GlobalQuit := FALSE;
   BB1_RZP2.Quit_RST := FALSE;
   BB1_RZP2.Tmr_VZ_Anlauf := 0;
   BB1_RZP2.Tmr_VZ_ESZ := 0;
   BB1_RZP2.Tmr_Th_St := 0;
   BB1_RZP2.Tmr_DMA_St := 0;
   BB1_RZP2.Tmr_DMZ_St := 0;
   BB1_RZP2.Tmr_FU_St := 0;
   BB1_RZP2.Tmr_TL_St := 0;
   BB1_RZP2.Tmr_UDr_St := 0;
   BB1_RZP2.Tmr_UeDr_St := 0;
   BB1_RZP2.Tmr_UT_St := 0;
   BB1_RZP2.Tmr_Le_St := 0;
   BB1_RZP2.Tmr_UeLM_St := 0;
   BB1_RZP2.Tmr_UeLE_St := 0;
   BB1_RZP2.Tmr_Kom_DP_St := 0;
   BB1_RZP2.Tmr_Kom_int_St := 0;
   BB1_RZP2.Tmr_int_St := 0;
   BB1_RZP2.Tmr_LZ_St := 0;
   BB1_RZP2.Tmr_BefLZ_St := 0;
   BB1_RZP2.Tmr_ASZ_St1 := 0;
   BB1_RZP2.Tmr_ASZ_St2 := 0;
   BB1_RZP2.Tmr_Rev_St1 := 0;
   BB1_RZP2.Tmr_Rev_St2 := 0;
   BB1_RZP2.BZ_ges_s := 2591;
   BB1_RZP2.Tmr_Quit_RST := 0;
   BB1_RZP2.BEF_NHV.Bef.Bed_Res := FALSE;
   BB1_RZP2.BEF_NHV.Bef.Bed_UV := FALSE;
   BB1_RZP2.BEF_NHV.Bef.Bed_NHV := FALSE;
   BB1_RZP2.BEF_NHV.Bef.Bed_PLS := FALSE;
   BB1_RZP2.BEF_NHV.Bef.BA_Hand := FALSE;
   BB1_RZP2.BEF_NHV.Bef.BA_Auto := FALSE;
   BB1_RZP2.BEF_NHV.Bef.BF_Ein1 := FALSE;
   BB1_RZP2.BEF_NHV.Bef.BF_Ein2 := FALSE;
   BB1_RZP2.BEF_NHV.Bef.BF_Aus := FALSE;
   BB1_RZP2.BEF_NHV.Bef.BZ_Res := FALSE;
   BB1_RZP2.BEF_NHV.Bef.Res_10 := FALSE;
   BB1_RZP2.BEF_NHV.Bef.Res_11 := FALSE;
   BB1_RZP2.BEF_NHV.Bef.Res_12 := FALSE;
   BB1_RZP2.BEF_NHV.Bef.Res_13 := FALSE;
   BB1_RZP2.BEF_NHV.Bef.Res_14 := FALSE;
   BB1_RZP2.BEF_NHV.Bef.Res_15 := FALSE;
   BB1_RZP2.BEF_NHV.Bef.Res_16 := FALSE;
   BB1_RZP2.BEF_NHV.Bef.Res_17 := FALSE;
   BB1_RZP2.BEF_NHV.Bef.Res_18 := FALSE;
   BB1_RZP2.BEF_NHV.Bef.Res_19 := FALSE;
   BB1_RZP2.BEF_NHV.Bef.Res_20 := FALSE;
   BB1_RZP2.BEF_NHV.Bef.Res_21 := FALSE;
   BB1_RZP2.BEF_NHV.Bef.Res_22 := FALSE;
   BB1_RZP2.BEF_NHV.Bef.Res_23 := FALSE;
   BB1_RZP2.BEF_NHV.Bef.Res_24 := FALSE;
   BB1_RZP2.BEF_NHV.Bef.Res_25 := FALSE;
   BB1_RZP2.BEF_NHV.Bef.Res_26 := FALSE;
   BB1_RZP2.BEF_NHV.Bef.Res_27 := FALSE;
   BB1_RZP2.BEF_NHV.Bef.Res_28 := FALSE;
   BB1_RZP2.BEF_NHV.Bef.Res_29 := FALSE;
   BB1_RZP2.BEF_NHV.Bef.BF_Set_SW_chg := FALSE;
   BB1_RZP2.BEF_NHV.Bef.BF_Quit := FALSE;
   BB1_RZP2.BEF_NHV.SW_Hand := 0.0;
   BB1_UeSP.Typ := 0;
   BB1_UeSP.Idx := 11;
   BB1_UeSP.BA_VW_Hand := FALSE;
   BB1_UeSP.Tmr_VZ_Anlauf_Q := FALSE;
   BB1_UeSP.SS := FALSE;
   BB1_UeSP.SSnq := FALSE;
   BB1_UeSP.SSfq := TRUE;
   BB1_UeSP.nBB := FALSE;
   BB1_UeSP.VW_Hand_St1 := FALSE;
   BB1_UeSP.VW_Hand_St2 := FALSE;
   BB1_UeSP.VW_Hand_Stop := FALSE;
   BB1_UeSP.VW_Auto_St1 := FALSE;
   BB1_UeSP.VW_Auto_St2 := FALSE;
   BB1_UeSP.Anst_Req_St1 := FALSE;
   BB1_UeSP.Anst_Req_St2 := FALSE;
   BB1_UeSP.FM_Betrieb_Ein := FALSE;
   BB1_UeSP.FM_Betrieb_Aus := TRUE;
   BB1_UeSP.NLZ_MAZ_St1 := FALSE;
   BB1_UeSP.NLZ_MAZ_St2 := FALSE;
   BB1_UeSP.NLZ_Rev_SS_St1 := FALSE;
   BB1_UeSP.NLZ_Rev_SS_St2 := FALSE;
   BB1_UeSP.Th_St := FALSE;
   BB1_UeSP.DMA_St := FALSE;
   BB1_UeSP.DMZ_St := FALSE;
   BB1_UeSP.FU_St := FALSE;
   BB1_UeSP.TL_St := FALSE;
   BB1_UeSP.UDr_St := FALSE;
   BB1_UeSP.UeDr_St := FALSE;
   BB1_UeSP.UT_St := FALSE;
   BB1_UeSP.Le_St := FALSE;
   BB1_UeSP.UeLM_St := FALSE;
   BB1_UeSP.UeLE_St := FALSE;
   BB1_UeSP.Kom_DP_St := FALSE;
   BB1_UeSP.Kom_int_St := FALSE;
   BB1_UeSP.int_St := FALSE;
   BB1_UeSP.LZ_St := FALSE;
   BB1_UeSP.BefLZ_St := FALSE;
   BB1_UeSP.FM_GlobalQuit := FALSE;
   BB1_UeSP.Quit_RST := FALSE;
   BB1_UeSP.Tmr_VZ_Anlauf := 0;
   BB1_UeSP.Tmr_VZ_ESZ := 0;
   BB1_UeSP.Tmr_Th_St := 0;
   BB1_UeSP.Tmr_DMA_St := 0;
   BB1_UeSP.Tmr_DMZ_St := 0;
   BB1_UeSP.Tmr_FU_St := 0;
   BB1_UeSP.Tmr_TL_St := 0;
   BB1_UeSP.Tmr_UDr_St := 0;
   BB1_UeSP.Tmr_UeDr_St := 0;
   BB1_UeSP.Tmr_UT_St := 0;
   BB1_UeSP.Tmr_Le_St := 0;
   BB1_UeSP.Tmr_UeLM_St := 0;
   BB1_UeSP.Tmr_UeLE_St := 0;
   BB1_UeSP.Tmr_Kom_DP_St := 0;
   BB1_UeSP.Tmr_Kom_int_St := 0;
   BB1_UeSP.Tmr_int_St := 0;
   BB1_UeSP.Tmr_LZ_St := 0;
   BB1_UeSP.Tmr_BefLZ_St := 0;
   BB1_UeSP.Tmr_ASZ_St1 := 0;
   BB1_UeSP.Tmr_ASZ_St2 := 0;
   BB1_UeSP.Tmr_Rev_St1 := 0;
   BB1_UeSP.Tmr_Rev_St2 := 0;
   BB1_UeSP.BZ_ges_s := 2740;
   BB1_UeSP.Tmr_Quit_RST := 0;
   BB1_UeSP.BEF_NHV.Bef.Bed_Res := FALSE;
   BB1_UeSP.BEF_NHV.Bef.Bed_UV := FALSE;
   BB1_UeSP.BEF_NHV.Bef.Bed_NHV := FALSE;
   BB1_UeSP.BEF_NHV.Bef.Bed_PLS := FALSE;
   BB1_UeSP.BEF_NHV.Bef.BA_Hand := FALSE;
   BB1_UeSP.BEF_NHV.Bef.BA_Auto := FALSE;
   BB1_UeSP.BEF_NHV.Bef.BF_Ein1 := FALSE;
   BB1_UeSP.BEF_NHV.Bef.BF_Ein2 := FALSE;
   BB1_UeSP.BEF_NHV.Bef.BF_Aus := FALSE;
   BB1_UeSP.BEF_NHV.Bef.BZ_Res := FALSE;
   BB1_UeSP.BEF_NHV.Bef.Res_10 := FALSE;
   BB1_UeSP.BEF_NHV.Bef.Res_11 := FALSE;
   BB1_UeSP.BEF_NHV.Bef.Res_12 := FALSE;
   BB1_UeSP.BEF_NHV.Bef.Res_13 := FALSE;
   BB1_UeSP.BEF_NHV.Bef.Res_14 := FALSE;
   BB1_UeSP.BEF_NHV.Bef.Res_15 := FALSE;
   BB1_UeSP.BEF_NHV.Bef.Res_16 := FALSE;
   BB1_UeSP.BEF_NHV.Bef.Res_17 := FALSE;
   BB1_UeSP.BEF_NHV.Bef.Res_18 := FALSE;
   BB1_UeSP.BEF_NHV.Bef.Res_19 := FALSE;
   BB1_UeSP.BEF_NHV.Bef.Res_20 := FALSE;
   BB1_UeSP.BEF_NHV.Bef.Res_21 := FALSE;
   BB1_UeSP.BEF_NHV.Bef.Res_22 := FALSE;
   BB1_UeSP.BEF_NHV.Bef.Res_23 := FALSE;
   BB1_UeSP.BEF_NHV.Bef.Res_24 := FALSE;
   BB1_UeSP.BEF_NHV.Bef.Res_25 := FALSE;
   BB1_UeSP.BEF_NHV.Bef.Res_26 := FALSE;
   BB1_UeSP.BEF_NHV.Bef.Res_27 := FALSE;
   BB1_UeSP.BEF_NHV.Bef.Res_28 := FALSE;
   BB1_UeSP.BEF_NHV.Bef.Res_29 := FALSE;
   BB1_UeSP.BEF_NHV.Bef.BF_Set_SW_chg := FALSE;
   BB1_UeSP.BEF_NHV.Bef.BF_Quit := FALSE;
   BB1_UeSP.BEF_NHV.SW_Hand := 0.0;
   BB1_AS1.Typ := 5;
   BB1_AS1.Idx := 12;
   BB1_AS1.BA_VW_Hand := FALSE;
   BB1_AS1.Tmr_VZ_Anlauf_Q := FALSE;
   BB1_AS1.SS := FALSE;
   BB1_AS1.SSnq := FALSE;
   BB1_AS1.SSfq := TRUE;
   BB1_AS1.nBB := FALSE;
   BB1_AS1.VW_Hand_St1 := FALSE;
   BB1_AS1.VW_Hand_St2 := FALSE;
   BB1_AS1.VW_Hand_Stop := FALSE;
   BB1_AS1.VW_Auto_St1 := FALSE;
   BB1_AS1.VW_Auto_St2 := FALSE;
   BB1_AS1.Anst_Req_St1 := FALSE;
   BB1_AS1.Anst_Req_St2 := FALSE;
   BB1_AS1.FM_Betrieb_Ein := FALSE;
   BB1_AS1.FM_Betrieb_Aus := TRUE;
   BB1_AS1.NLZ_MAZ_St1 := FALSE;
   BB1_AS1.NLZ_MAZ_St2 := FALSE;
   BB1_AS1.NLZ_Rev_SS_St1 := FALSE;
   BB1_AS1.NLZ_Rev_SS_St2 := FALSE;
   BB1_AS1.Th_St := FALSE;
   BB1_AS1.DMA_St := FALSE;
   BB1_AS1.DMZ_St := FALSE;
   BB1_AS1.FU_St := FALSE;
   BB1_AS1.TL_St := FALSE;
   BB1_AS1.UDr_St := FALSE;
   BB1_AS1.UeDr_St := FALSE;
   BB1_AS1.UT_St := FALSE;
   BB1_AS1.Le_St := FALSE;
   BB1_AS1.UeLM_St := FALSE;
   BB1_AS1.UeLE_St := FALSE;
   BB1_AS1.Kom_DP_St := FALSE;
   BB1_AS1.Kom_int_St := FALSE;
   BB1_AS1.int_St := FALSE;
   BB1_AS1.LZ_St := FALSE;
   BB1_AS1.BefLZ_St := FALSE;
   BB1_AS1.FM_GlobalQuit := FALSE;
   BB1_AS1.Quit_RST := FALSE;
   BB1_AS1.Tmr_VZ_Anlauf := 0;
   BB1_AS1.Tmr_VZ_ESZ := 0;
   BB1_AS1.Tmr_Th_St := 0;
   BB1_AS1.Tmr_DMA_St := 0;
   BB1_AS1.Tmr_DMZ_St := 0;
   BB1_AS1.Tmr_FU_St := 0;
   BB1_AS1.Tmr_TL_St := 0;
   BB1_AS1.Tmr_UDr_St := 0;
   BB1_AS1.Tmr_UeDr_St := 0;
   BB1_AS1.Tmr_UT_St := 0;
   BB1_AS1.Tmr_Le_St := 0;
   BB1_AS1.Tmr_UeLM_St := 0;
   BB1_AS1.Tmr_UeLE_St := 0;
   BB1_AS1.Tmr_Kom_DP_St := 0;
   BB1_AS1.Tmr_Kom_int_St := 0;
   BB1_AS1.Tmr_int_St := 0;
   BB1_AS1.Tmr_LZ_St := 0;
   BB1_AS1.Tmr_BefLZ_St := 0;
   BB1_AS1.Tmr_ASZ_St1 := 0;
   BB1_AS1.Tmr_ASZ_St2 := 0;
   BB1_AS1.Tmr_Rev_St1 := 0;
   BB1_AS1.Tmr_Rev_St2 := 0;
   BB1_AS1.BZ_ges_s := 2050;
   BB1_AS1.Tmr_Quit_RST := 0;
   BB1_AS1.BEF_NHV.Bef.Bed_Res := FALSE;
   BB1_AS1.BEF_NHV.Bef.Bed_UV := FALSE;
   BB1_AS1.BEF_NHV.Bef.Bed_NHV := FALSE;
   BB1_AS1.BEF_NHV.Bef.Bed_PLS := FALSE;
   BB1_AS1.BEF_NHV.Bef.BA_Hand := FALSE;
   BB1_AS1.BEF_NHV.Bef.BA_Auto := FALSE;
   BB1_AS1.BEF_NHV.Bef.BF_Ein1 := FALSE;
   BB1_AS1.BEF_NHV.Bef.BF_Ein2 := FALSE;
   BB1_AS1.BEF_NHV.Bef.BF_Aus := FALSE;
   BB1_AS1.BEF_NHV.Bef.BZ_Res := FALSE;
   BB1_AS1.BEF_NHV.Bef.Res_10 := FALSE;
   BB1_AS1.BEF_NHV.Bef.Res_11 := FALSE;
   BB1_AS1.BEF_NHV.Bef.Res_12 := FALSE;
   BB1_AS1.BEF_NHV.Bef.Res_13 := FALSE;
   BB1_AS1.BEF_NHV.Bef.Res_14 := FALSE;
   BB1_AS1.BEF_NHV.Bef.Res_15 := FALSE;
   BB1_AS1.BEF_NHV.Bef.Res_16 := FALSE;
   BB1_AS1.BEF_NHV.Bef.Res_17 := FALSE;
   BB1_AS1.BEF_NHV.Bef.Res_18 := FALSE;
   BB1_AS1.BEF_NHV.Bef.Res_19 := FALSE;
   BB1_AS1.BEF_NHV.Bef.Res_20 := FALSE;
   BB1_AS1.BEF_NHV.Bef.Res_21 := FALSE;
   BB1_AS1.BEF_NHV.Bef.Res_22 := FALSE;
   BB1_AS1.BEF_NHV.Bef.Res_23 := FALSE;
   BB1_AS1.BEF_NHV.Bef.Res_24 := FALSE;
   BB1_AS1.BEF_NHV.Bef.Res_25 := FALSE;
   BB1_AS1.BEF_NHV.Bef.Res_26 := FALSE;
   BB1_AS1.BEF_NHV.Bef.Res_27 := FALSE;
   BB1_AS1.BEF_NHV.Bef.Res_28 := FALSE;
   BB1_AS1.BEF_NHV.Bef.Res_29 := FALSE;
   BB1_AS1.BEF_NHV.Bef.BF_Set_SW_chg := FALSE;
   BB1_AS1.BEF_NHV.Bef.BF_Quit := FALSE;
   BB1_AS1.BEF_NHV.SW_Hand := 0.0;
   BB1_AS2.Typ := 5;
   BB1_AS2.Idx := 13;
   BB1_AS2.BA_VW_Hand := FALSE;
   BB1_AS2.Tmr_VZ_Anlauf_Q := FALSE;
   BB1_AS2.SS := FALSE;
   BB1_AS2.SSnq := FALSE;
   BB1_AS2.SSfq := TRUE;
   BB1_AS2.nBB := FALSE;
   BB1_AS2.VW_Hand_St1 := FALSE;
   BB1_AS2.VW_Hand_St2 := FALSE;
   BB1_AS2.VW_Hand_Stop := FALSE;
   BB1_AS2.VW_Auto_St1 := FALSE;
   BB1_AS2.VW_Auto_St2 := FALSE;
   BB1_AS2.Anst_Req_St1 := FALSE;
   BB1_AS2.Anst_Req_St2 := FALSE;
   BB1_AS2.FM_Betrieb_Ein := FALSE;
   BB1_AS2.FM_Betrieb_Aus := TRUE;
   BB1_AS2.NLZ_MAZ_St1 := FALSE;
   BB1_AS2.NLZ_MAZ_St2 := FALSE;
   BB1_AS2.NLZ_Rev_SS_St1 := FALSE;
   BB1_AS2.NLZ_Rev_SS_St2 := FALSE;
   BB1_AS2.Th_St := FALSE;
   BB1_AS2.DMA_St := FALSE;
   BB1_AS2.DMZ_St := FALSE;
   BB1_AS2.FU_St := FALSE;
   BB1_AS2.TL_St := FALSE;
   BB1_AS2.UDr_St := FALSE;
   BB1_AS2.UeDr_St := FALSE;
   BB1_AS2.UT_St := FALSE;
   BB1_AS2.Le_St := FALSE;
   BB1_AS2.UeLM_St := FALSE;
   BB1_AS2.UeLE_St := FALSE;
   BB1_AS2.Kom_DP_St := FALSE;
   BB1_AS2.Kom_int_St := FALSE;
   BB1_AS2.int_St := FALSE;
   BB1_AS2.LZ_St := FALSE;
   BB1_AS2.BefLZ_St := FALSE;
   BB1_AS2.FM_GlobalQuit := FALSE;
   BB1_AS2.Quit_RST := FALSE;
   BB1_AS2.Tmr_VZ_Anlauf := 0;
   BB1_AS2.Tmr_VZ_ESZ := 0;
   BB1_AS2.Tmr_Th_St := 0;
   BB1_AS2.Tmr_DMA_St := 0;
   BB1_AS2.Tmr_DMZ_St := 0;
   BB1_AS2.Tmr_FU_St := 0;
   BB1_AS2.Tmr_TL_St := 0;
   BB1_AS2.Tmr_UDr_St := 0;
   BB1_AS2.Tmr_UeDr_St := 0;
   BB1_AS2.Tmr_UT_St := 0;
   BB1_AS2.Tmr_Le_St := 0;
   BB1_AS2.Tmr_UeLM_St := 0;
   BB1_AS2.Tmr_UeLE_St := 0;
   BB1_AS2.Tmr_Kom_DP_St := 0;
   BB1_AS2.Tmr_Kom_int_St := 0;
   BB1_AS2.Tmr_int_St := 0;
   BB1_AS2.Tmr_LZ_St := 0;
   BB1_AS2.Tmr_BefLZ_St := 0;
   BB1_AS2.Tmr_ASZ_St1 := 0;
   BB1_AS2.Tmr_ASZ_St2 := 0;
   BB1_AS2.Tmr_Rev_St1 := 0;
   BB1_AS2.Tmr_Rev_St2 := 0;
   BB1_AS2.BZ_ges_s := 1084;
   BB1_AS2.Tmr_Quit_RST := 0;
   BB1_AS2.BEF_NHV.Bef.Bed_Res := FALSE;
   BB1_AS2.BEF_NHV.Bef.Bed_UV := FALSE;
   BB1_AS2.BEF_NHV.Bef.Bed_NHV := FALSE;
   BB1_AS2.BEF_NHV.Bef.Bed_PLS := FALSE;
   BB1_AS2.BEF_NHV.Bef.BA_Hand := FALSE;
   BB1_AS2.BEF_NHV.Bef.BA_Auto := FALSE;
   BB1_AS2.BEF_NHV.Bef.BF_Ein1 := FALSE;
   BB1_AS2.BEF_NHV.Bef.BF_Ein2 := FALSE;
   BB1_AS2.BEF_NHV.Bef.BF_Aus := FALSE;
   BB1_AS2.BEF_NHV.Bef.BZ_Res := FALSE;
   BB1_AS2.BEF_NHV.Bef.Res_10 := FALSE;
   BB1_AS2.BEF_NHV.Bef.Res_11 := FALSE;
   BB1_AS2.BEF_NHV.Bef.Res_12 := FALSE;
   BB1_AS2.BEF_NHV.Bef.Res_13 := FALSE;
   BB1_AS2.BEF_NHV.Bef.Res_14 := FALSE;
   BB1_AS2.BEF_NHV.Bef.Res_15 := FALSE;
   BB1_AS2.BEF_NHV.Bef.Res_16 := FALSE;
   BB1_AS2.BEF_NHV.Bef.Res_17 := FALSE;
   BB1_AS2.BEF_NHV.Bef.Res_18 := FALSE;
   BB1_AS2.BEF_NHV.Bef.Res_19 := FALSE;
   BB1_AS2.BEF_NHV.Bef.Res_20 := FALSE;
   BB1_AS2.BEF_NHV.Bef.Res_21 := FALSE;
   BB1_AS2.BEF_NHV.Bef.Res_22 := FALSE;
   BB1_AS2.BEF_NHV.Bef.Res_23 := FALSE;
   BB1_AS2.BEF_NHV.Bef.Res_24 := FALSE;
   BB1_AS2.BEF_NHV.Bef.Res_25 := FALSE;
   BB1_AS2.BEF_NHV.Bef.Res_26 := FALSE;
   BB1_AS2.BEF_NHV.Bef.Res_27 := FALSE;
   BB1_AS2.BEF_NHV.Bef.Res_28 := FALSE;
   BB1_AS2.BEF_NHV.Bef.Res_29 := FALSE;
   BB1_AS2.BEF_NHV.Bef.BF_Set_SW_chg := FALSE;
   BB1_AS2.BEF_NHV.Bef.BF_Quit := FALSE;
   BB1_AS2.BEF_NHV.SW_Hand := 0.0;
   BB1_SR1.Typ := 7;
   BB1_SR1.Idx := 14;
   BB1_SR1.BA_VW_Hand := FALSE;
   BB1_SR1.Tmr_VZ_Anlauf_Q := FALSE;
   BB1_SR1.SS := FALSE;
   BB1_SR1.SSnq := FALSE;
   BB1_SR1.SSfq := TRUE;
   BB1_SR1.nBB := FALSE;
   BB1_SR1.VW_Hand_St1 := FALSE;
   BB1_SR1.VW_Hand_St2 := FALSE;
   BB1_SR1.VW_Hand_Stop := FALSE;
   BB1_SR1.VW_Auto_St1 := FALSE;
   BB1_SR1.VW_Auto_St2 := FALSE;
   BB1_SR1.Anst_Req_St1 := FALSE;
   BB1_SR1.Anst_Req_St2 := FALSE;
   BB1_SR1.FM_Betrieb_Ein := FALSE;
   BB1_SR1.FM_Betrieb_Aus := TRUE;
   BB1_SR1.NLZ_MAZ_St1 := FALSE;
   BB1_SR1.NLZ_MAZ_St2 := FALSE;
   BB1_SR1.NLZ_Rev_SS_St1 := FALSE;
   BB1_SR1.NLZ_Rev_SS_St2 := FALSE;
   BB1_SR1.Th_St := FALSE;
   BB1_SR1.DMA_St := FALSE;
   BB1_SR1.DMZ_St := FALSE;
   BB1_SR1.FU_St := FALSE;
   BB1_SR1.TL_St := FALSE;
   BB1_SR1.UDr_St := FALSE;
   BB1_SR1.UeDr_St := FALSE;
   BB1_SR1.UT_St := FALSE;
   BB1_SR1.Le_St := FALSE;
   BB1_SR1.UeLM_St := FALSE;
   BB1_SR1.UeLE_St := FALSE;
   BB1_SR1.Kom_DP_St := FALSE;
   BB1_SR1.Kom_int_St := FALSE;
   BB1_SR1.int_St := FALSE;
   BB1_SR1.LZ_St := FALSE;
   BB1_SR1.BefLZ_St := FALSE;
   BB1_SR1.FM_GlobalQuit := FALSE;
   BB1_SR1.Quit_RST := FALSE;
   BB1_SR1.Tmr_VZ_Anlauf := 0;
   BB1_SR1.Tmr_VZ_ESZ := 0;
   BB1_SR1.Tmr_Th_St := 0;
   BB1_SR1.Tmr_DMA_St := 0;
   BB1_SR1.Tmr_DMZ_St := 0;
   BB1_SR1.Tmr_FU_St := 0;
   BB1_SR1.Tmr_TL_St := 0;
   BB1_SR1.Tmr_UDr_St := 0;
   BB1_SR1.Tmr_UeDr_St := 0;
   BB1_SR1.Tmr_UT_St := 0;
   BB1_SR1.Tmr_Le_St := 0;
   BB1_SR1.Tmr_UeLM_St := 0;
   BB1_SR1.Tmr_UeLE_St := 0;
   BB1_SR1.Tmr_Kom_DP_St := 0;
   BB1_SR1.Tmr_Kom_int_St := 0;
   BB1_SR1.Tmr_int_St := 0;
   BB1_SR1.Tmr_LZ_St := 0;
   BB1_SR1.Tmr_BefLZ_St := 0;
   BB1_SR1.Tmr_ASZ_St1 := 0;
   BB1_SR1.Tmr_ASZ_St2 := 0;
   BB1_SR1.Tmr_Rev_St1 := 0;
   BB1_SR1.Tmr_Rev_St2 := 0;
   BB1_SR1.BZ_ges_s := 2705;
   BB1_SR1.Tmr_Quit_RST := 0;
   BB1_SR1.BEF_NHV.Bef.Bed_Res := FALSE;
   BB1_SR1.BEF_NHV.Bef.Bed_UV := FALSE;
   BB1_SR1.BEF_NHV.Bef.Bed_NHV := FALSE;
   BB1_SR1.BEF_NHV.Bef.Bed_PLS := FALSE;
   BB1_SR1.BEF_NHV.Bef.BA_Hand := FALSE;
   BB1_SR1.BEF_NHV.Bef.BA_Auto := FALSE;
   BB1_SR1.BEF_NHV.Bef.BF_Ein1 := FALSE;
   BB1_SR1.BEF_NHV.Bef.BF_Ein2 := FALSE;
   BB1_SR1.BEF_NHV.Bef.BF_Aus := FALSE;
   BB1_SR1.BEF_NHV.Bef.BZ_Res := FALSE;
   BB1_SR1.BEF_NHV.Bef.Res_10 := FALSE;
   BB1_SR1.BEF_NHV.Bef.Res_11 := FALSE;
   BB1_SR1.BEF_NHV.Bef.Res_12 := FALSE;
   BB1_SR1.BEF_NHV.Bef.Res_13 := FALSE;
   BB1_SR1.BEF_NHV.Bef.Res_14 := FALSE;
   BB1_SR1.BEF_NHV.Bef.Res_15 := FALSE;
   BB1_SR1.BEF_NHV.Bef.Res_16 := FALSE;
   BB1_SR1.BEF_NHV.Bef.Res_17 := FALSE;
   BB1_SR1.BEF_NHV.Bef.Res_18 := FALSE;
   BB1_SR1.BEF_NHV.Bef.Res_19 := FALSE;
   BB1_SR1.BEF_NHV.Bef.Res_20 := FALSE;
   BB1_SR1.BEF_NHV.Bef.Res_21 := FALSE;
   BB1_SR1.BEF_NHV.Bef.Res_22 := FALSE;
   BB1_SR1.BEF_NHV.Bef.Res_23 := FALSE;
   BB1_SR1.BEF_NHV.Bef.Res_24 := FALSE;
   BB1_SR1.BEF_NHV.Bef.Res_25 := FALSE;
   BB1_SR1.BEF_NHV.Bef.Res_26 := FALSE;
   BB1_SR1.BEF_NHV.Bef.Res_27 := FALSE;
   BB1_SR1.BEF_NHV.Bef.Res_28 := FALSE;
   BB1_SR1.BEF_NHV.Bef.Res_29 := FALSE;
   BB1_SR1.BEF_NHV.Bef.BF_Set_SW_chg := FALSE;
   BB1_SR1.BEF_NHV.Bef.BF_Quit := FALSE;
   BB1_SR1.BEF_NHV.SW_Hand := 0.0;
   BB1_SR2.Typ := 7;
   BB1_SR2.Idx := 15;
   BB1_SR2.BA_VW_Hand := FALSE;
   BB1_SR2.Tmr_VZ_Anlauf_Q := FALSE;
   BB1_SR2.SS := FALSE;
   BB1_SR2.SSnq := FALSE;
   BB1_SR2.SSfq := TRUE;
   BB1_SR2.nBB := FALSE;
   BB1_SR2.VW_Hand_St1 := FALSE;
   BB1_SR2.VW_Hand_St2 := FALSE;
   BB1_SR2.VW_Hand_Stop := FALSE;
   BB1_SR2.VW_Auto_St1 := FALSE;
   BB1_SR2.VW_Auto_St2 := FALSE;
   BB1_SR2.Anst_Req_St1 := FALSE;
   BB1_SR2.Anst_Req_St2 := FALSE;
   BB1_SR2.FM_Betrieb_Ein := FALSE;
   BB1_SR2.FM_Betrieb_Aus := TRUE;
   BB1_SR2.NLZ_MAZ_St1 := FALSE;
   BB1_SR2.NLZ_MAZ_St2 := FALSE;
   BB1_SR2.NLZ_Rev_SS_St1 := FALSE;
   BB1_SR2.NLZ_Rev_SS_St2 := FALSE;
   BB1_SR2.Th_St := FALSE;
   BB1_SR2.DMA_St := FALSE;
   BB1_SR2.DMZ_St := FALSE;
   BB1_SR2.FU_St := FALSE;
   BB1_SR2.TL_St := FALSE;
   BB1_SR2.UDr_St := FALSE;
   BB1_SR2.UeDr_St := FALSE;
   BB1_SR2.UT_St := FALSE;
   BB1_SR2.Le_St := FALSE;
   BB1_SR2.UeLM_St := FALSE;
   BB1_SR2.UeLE_St := FALSE;
   BB1_SR2.Kom_DP_St := FALSE;
   BB1_SR2.Kom_int_St := FALSE;
   BB1_SR2.int_St := FALSE;
   BB1_SR2.LZ_St := FALSE;
   BB1_SR2.BefLZ_St := FALSE;
   BB1_SR2.FM_GlobalQuit := FALSE;
   BB1_SR2.Quit_RST := FALSE;
   BB1_SR2.Tmr_VZ_Anlauf := 0;
   BB1_SR2.Tmr_VZ_ESZ := 0;
   BB1_SR2.Tmr_Th_St := 0;
   BB1_SR2.Tmr_DMA_St := 0;
   BB1_SR2.Tmr_DMZ_St := 0;
   BB1_SR2.Tmr_FU_St := 0;
   BB1_SR2.Tmr_TL_St := 0;
   BB1_SR2.Tmr_UDr_St := 0;
   BB1_SR2.Tmr_UeDr_St := 0;
   BB1_SR2.Tmr_UT_St := 0;
   BB1_SR2.Tmr_Le_St := 0;
   BB1_SR2.Tmr_UeLM_St := 0;
   BB1_SR2.Tmr_UeLE_St := 0;
   BB1_SR2.Tmr_Kom_DP_St := 0;
   BB1_SR2.Tmr_Kom_int_St := 0;
   BB1_SR2.Tmr_int_St := 0;
   BB1_SR2.Tmr_LZ_St := 0;
   BB1_SR2.Tmr_BefLZ_St := 0;
   BB1_SR2.Tmr_ASZ_St1 := 0;
   BB1_SR2.Tmr_ASZ_St2 := 0;
   BB1_SR2.Tmr_Rev_St1 := 0;
   BB1_SR2.Tmr_Rev_St2 := 0;
   BB1_SR2.BZ_ges_s := 2698;
   BB1_SR2.Tmr_Quit_RST := 0;
   BB1_SR2.BEF_NHV.Bef.Bed_Res := FALSE;
   BB1_SR2.BEF_NHV.Bef.Bed_UV := FALSE;
   BB1_SR2.BEF_NHV.Bef.Bed_NHV := FALSE;
   BB1_SR2.BEF_NHV.Bef.Bed_PLS := FALSE;
   BB1_SR2.BEF_NHV.Bef.BA_Hand := FALSE;
   BB1_SR2.BEF_NHV.Bef.BA_Auto := FALSE;
   BB1_SR2.BEF_NHV.Bef.BF_Ein1 := FALSE;
   BB1_SR2.BEF_NHV.Bef.BF_Ein2 := FALSE;
   BB1_SR2.BEF_NHV.Bef.BF_Aus := FALSE;
   BB1_SR2.BEF_NHV.Bef.BZ_Res := FALSE;
   BB1_SR2.BEF_NHV.Bef.Res_10 := FALSE;
   BB1_SR2.BEF_NHV.Bef.Res_11 := FALSE;
   BB1_SR2.BEF_NHV.Bef.Res_12 := FALSE;
   BB1_SR2.BEF_NHV.Bef.Res_13 := FALSE;
   BB1_SR2.BEF_NHV.Bef.Res_14 := FALSE;
   BB1_SR2.BEF_NHV.Bef.Res_15 := FALSE;
   BB1_SR2.BEF_NHV.Bef.Res_16 := FALSE;
   BB1_SR2.BEF_NHV.Bef.Res_17 := FALSE;
   BB1_SR2.BEF_NHV.Bef.Res_18 := FALSE;
   BB1_SR2.BEF_NHV.Bef.Res_19 := FALSE;
   BB1_SR2.BEF_NHV.Bef.Res_20 := FALSE;
   BB1_SR2.BEF_NHV.Bef.Res_21 := FALSE;
   BB1_SR2.BEF_NHV.Bef.Res_22 := FALSE;
   BB1_SR2.BEF_NHV.Bef.Res_23 := FALSE;
   BB1_SR2.BEF_NHV.Bef.Res_24 := FALSE;
   BB1_SR2.BEF_NHV.Bef.Res_25 := FALSE;
   BB1_SR2.BEF_NHV.Bef.Res_26 := FALSE;
   BB1_SR2.BEF_NHV.Bef.Res_27 := FALSE;
   BB1_SR2.BEF_NHV.Bef.Res_28 := FALSE;
   BB1_SR2.BEF_NHV.Bef.Res_29 := FALSE;
   BB1_SR2.BEF_NHV.Bef.BF_Set_SW_chg := FALSE;
   BB1_SR2.BEF_NHV.Bef.BF_Quit := FALSE;
   BB1_SR2.BEF_NHV.SW_Hand := 0.0;
   BB2_RZP1.Typ := 0;
   BB2_RZP1.Idx := 16;
   BB2_RZP1.BA_VW_Hand := FALSE;
   BB2_RZP1.Tmr_VZ_Anlauf_Q := FALSE;
   BB2_RZP1.SS := FALSE;
   BB2_RZP1.SSnq := FALSE;
   BB2_RZP1.SSfq := TRUE;
   BB2_RZP1.nBB := FALSE;
   BB2_RZP1.VW_Hand_St1 := FALSE;
   BB2_RZP1.VW_Hand_St2 := FALSE;
   BB2_RZP1.VW_Hand_Stop := FALSE;
   BB2_RZP1.VW_Auto_St1 := FALSE;
   BB2_RZP1.VW_Auto_St2 := FALSE;
   BB2_RZP1.Anst_Req_St1 := FALSE;
   BB2_RZP1.Anst_Req_St2 := FALSE;
   BB2_RZP1.FM_Betrieb_Ein := FALSE;
   BB2_RZP1.FM_Betrieb_Aus := TRUE;
   BB2_RZP1.NLZ_MAZ_St1 := FALSE;
   BB2_RZP1.NLZ_MAZ_St2 := FALSE;
   BB2_RZP1.NLZ_Rev_SS_St1 := FALSE;
   BB2_RZP1.NLZ_Rev_SS_St2 := FALSE;
   BB2_RZP1.Th_St := FALSE;
   BB2_RZP1.DMA_St := FALSE;
   BB2_RZP1.DMZ_St := FALSE;
   BB2_RZP1.FU_St := FALSE;
   BB2_RZP1.TL_St := FALSE;
   BB2_RZP1.UDr_St := FALSE;
   BB2_RZP1.UeDr_St := FALSE;
   BB2_RZP1.UT_St := FALSE;
   BB2_RZP1.Le_St := FALSE;
   BB2_RZP1.UeLM_St := FALSE;
   BB2_RZP1.UeLE_St := FALSE;
   BB2_RZP1.Kom_DP_St := FALSE;
   BB2_RZP1.Kom_int_St := FALSE;
   BB2_RZP1.int_St := FALSE;
   BB2_RZP1.LZ_St := FALSE;
   BB2_RZP1.BefLZ_St := FALSE;
   BB2_RZP1.FM_GlobalQuit := FALSE;
   BB2_RZP1.Quit_RST := FALSE;
   BB2_RZP1.Tmr_VZ_Anlauf := 0;
   BB2_RZP1.Tmr_VZ_ESZ := 0;
   BB2_RZP1.Tmr_Th_St := 0;
   BB2_RZP1.Tmr_DMA_St := 0;
   BB2_RZP1.Tmr_DMZ_St := 0;
   BB2_RZP1.Tmr_FU_St := 0;
   BB2_RZP1.Tmr_TL_St := 0;
   BB2_RZP1.Tmr_UDr_St := 0;
   BB2_RZP1.Tmr_UeDr_St := 0;
   BB2_RZP1.Tmr_UT_St := 0;
   BB2_RZP1.Tmr_Le_St := 0;
   BB2_RZP1.Tmr_UeLM_St := 0;
   BB2_RZP1.Tmr_UeLE_St := 0;
   BB2_RZP1.Tmr_Kom_DP_St := 0;
   BB2_RZP1.Tmr_Kom_int_St := 0;
   BB2_RZP1.Tmr_int_St := 0;
   BB2_RZP1.Tmr_LZ_St := 0;
   BB2_RZP1.Tmr_BefLZ_St := 0;
   BB2_RZP1.Tmr_ASZ_St1 := 0;
   BB2_RZP1.Tmr_ASZ_St2 := 0;
   BB2_RZP1.Tmr_Rev_St1 := 0;
   BB2_RZP1.Tmr_Rev_St2 := 0;
   BB2_RZP1.BZ_ges_s := 2197;
   BB2_RZP1.Tmr_Quit_RST := 0;
   BB2_RZP1.BEF_NHV.Bef.Bed_Res := FALSE;
   BB2_RZP1.BEF_NHV.Bef.Bed_UV := FALSE;
   BB2_RZP1.BEF_NHV.Bef.Bed_NHV := FALSE;
   BB2_RZP1.BEF_NHV.Bef.Bed_PLS := FALSE;
   BB2_RZP1.BEF_NHV.Bef.BA_Hand := FALSE;
   BB2_RZP1.BEF_NHV.Bef.BA_Auto := FALSE;
   BB2_RZP1.BEF_NHV.Bef.BF_Ein1 := FALSE;
   BB2_RZP1.BEF_NHV.Bef.BF_Ein2 := FALSE;
   BB2_RZP1.BEF_NHV.Bef.BF_Aus := FALSE;
   BB2_RZP1.BEF_NHV.Bef.BZ_Res := FALSE;
   BB2_RZP1.BEF_NHV.Bef.Res_10 := FALSE;
   BB2_RZP1.BEF_NHV.Bef.Res_11 := FALSE;
   BB2_RZP1.BEF_NHV.Bef.Res_12 := FALSE;
   BB2_RZP1.BEF_NHV.Bef.Res_13 := FALSE;
   BB2_RZP1.BEF_NHV.Bef.Res_14 := FALSE;
   BB2_RZP1.BEF_NHV.Bef.Res_15 := FALSE;
   BB2_RZP1.BEF_NHV.Bef.Res_16 := FALSE;
   BB2_RZP1.BEF_NHV.Bef.Res_17 := FALSE;
   BB2_RZP1.BEF_NHV.Bef.Res_18 := FALSE;
   BB2_RZP1.BEF_NHV.Bef.Res_19 := FALSE;
   BB2_RZP1.BEF_NHV.Bef.Res_20 := FALSE;
   BB2_RZP1.BEF_NHV.Bef.Res_21 := FALSE;
   BB2_RZP1.BEF_NHV.Bef.Res_22 := FALSE;
   BB2_RZP1.BEF_NHV.Bef.Res_23 := FALSE;
   BB2_RZP1.BEF_NHV.Bef.Res_24 := FALSE;
   BB2_RZP1.BEF_NHV.Bef.Res_25 := FALSE;
   BB2_RZP1.BEF_NHV.Bef.Res_26 := FALSE;
   BB2_RZP1.BEF_NHV.Bef.Res_27 := FALSE;
   BB2_RZP1.BEF_NHV.Bef.Res_28 := FALSE;
   BB2_RZP1.BEF_NHV.Bef.Res_29 := FALSE;
   BB2_RZP1.BEF_NHV.Bef.BF_Set_SW_chg := FALSE;
   BB2_RZP1.BEF_NHV.Bef.BF_Quit := FALSE;
   BB2_RZP1.BEF_NHV.SW_Hand := 0.0;
   BB2_RZP2.Typ := 0;
   BB2_RZP2.Idx := 17;
   BB2_RZP2.BA_VW_Hand := FALSE;
   BB2_RZP2.Tmr_VZ_Anlauf_Q := FALSE;
   BB2_RZP2.SS := FALSE;
   BB2_RZP2.SSnq := FALSE;
   BB2_RZP2.SSfq := TRUE;
   BB2_RZP2.nBB := FALSE;
   BB2_RZP2.VW_Hand_St1 := FALSE;
   BB2_RZP2.VW_Hand_St2 := FALSE;
   BB2_RZP2.VW_Hand_Stop := FALSE;
   BB2_RZP2.VW_Auto_St1 := FALSE;
   BB2_RZP2.VW_Auto_St2 := FALSE;
   BB2_RZP2.Anst_Req_St1 := FALSE;
   BB2_RZP2.Anst_Req_St2 := FALSE;
   BB2_RZP2.FM_Betrieb_Ein := FALSE;
   BB2_RZP2.FM_Betrieb_Aus := TRUE;
   BB2_RZP2.NLZ_MAZ_St1 := FALSE;
   BB2_RZP2.NLZ_MAZ_St2 := FALSE;
   BB2_RZP2.NLZ_Rev_SS_St1 := FALSE;
   BB2_RZP2.NLZ_Rev_SS_St2 := FALSE;
   BB2_RZP2.Th_St := FALSE;
   BB2_RZP2.DMA_St := FALSE;
   BB2_RZP2.DMZ_St := FALSE;
   BB2_RZP2.FU_St := FALSE;
   BB2_RZP2.TL_St := FALSE;
   BB2_RZP2.UDr_St := FALSE;
   BB2_RZP2.UeDr_St := FALSE;
   BB2_RZP2.UT_St := FALSE;
   BB2_RZP2.Le_St := FALSE;
   BB2_RZP2.UeLM_St := FALSE;
   BB2_RZP2.UeLE_St := FALSE;
   BB2_RZP2.Kom_DP_St := FALSE;
   BB2_RZP2.Kom_int_St := FALSE;
   BB2_RZP2.int_St := FALSE;
   BB2_RZP2.LZ_St := FALSE;
   BB2_RZP2.BefLZ_St := FALSE;
   BB2_RZP2.FM_GlobalQuit := FALSE;
   BB2_RZP2.Quit_RST := FALSE;
   BB2_RZP2.Tmr_VZ_Anlauf := 0;
   BB2_RZP2.Tmr_VZ_ESZ := 0;
   BB2_RZP2.Tmr_Th_St := 0;
   BB2_RZP2.Tmr_DMA_St := 0;
   BB2_RZP2.Tmr_DMZ_St := 0;
   BB2_RZP2.Tmr_FU_St := 0;
   BB2_RZP2.Tmr_TL_St := 0;
   BB2_RZP2.Tmr_UDr_St := 0;
   BB2_RZP2.Tmr_UeDr_St := 0;
   BB2_RZP2.Tmr_UT_St := 0;
   BB2_RZP2.Tmr_Le_St := 0;
   BB2_RZP2.Tmr_UeLM_St := 0;
   BB2_RZP2.Tmr_UeLE_St := 0;
   BB2_RZP2.Tmr_Kom_DP_St := 0;
   BB2_RZP2.Tmr_Kom_int_St := 0;
   BB2_RZP2.Tmr_int_St := 0;
   BB2_RZP2.Tmr_LZ_St := 0;
   BB2_RZP2.Tmr_BefLZ_St := 0;
   BB2_RZP2.Tmr_ASZ_St1 := 0;
   BB2_RZP2.Tmr_ASZ_St2 := 0;
   BB2_RZP2.Tmr_Rev_St1 := 0;
   BB2_RZP2.Tmr_Rev_St2 := 0;
   BB2_RZP2.BZ_ges_s := 2494;
   BB2_RZP2.Tmr_Quit_RST := 0;
   BB2_RZP2.BEF_NHV.Bef.Bed_Res := FALSE;
   BB2_RZP2.BEF_NHV.Bef.Bed_UV := FALSE;
   BB2_RZP2.BEF_NHV.Bef.Bed_NHV := FALSE;
   BB2_RZP2.BEF_NHV.Bef.Bed_PLS := FALSE;
   BB2_RZP2.BEF_NHV.Bef.BA_Hand := FALSE;
   BB2_RZP2.BEF_NHV.Bef.BA_Auto := FALSE;
   BB2_RZP2.BEF_NHV.Bef.BF_Ein1 := FALSE;
   BB2_RZP2.BEF_NHV.Bef.BF_Ein2 := FALSE;
   BB2_RZP2.BEF_NHV.Bef.BF_Aus := FALSE;
   BB2_RZP2.BEF_NHV.Bef.BZ_Res := FALSE;
   BB2_RZP2.BEF_NHV.Bef.Res_10 := FALSE;
   BB2_RZP2.BEF_NHV.Bef.Res_11 := FALSE;
   BB2_RZP2.BEF_NHV.Bef.Res_12 := FALSE;
   BB2_RZP2.BEF_NHV.Bef.Res_13 := FALSE;
   BB2_RZP2.BEF_NHV.Bef.Res_14 := FALSE;
   BB2_RZP2.BEF_NHV.Bef.Res_15 := FALSE;
   BB2_RZP2.BEF_NHV.Bef.Res_16 := FALSE;
   BB2_RZP2.BEF_NHV.Bef.Res_17 := FALSE;
   BB2_RZP2.BEF_NHV.Bef.Res_18 := FALSE;
   BB2_RZP2.BEF_NHV.Bef.Res_19 := FALSE;
   BB2_RZP2.BEF_NHV.Bef.Res_20 := FALSE;
   BB2_RZP2.BEF_NHV.Bef.Res_21 := FALSE;
   BB2_RZP2.BEF_NHV.Bef.Res_22 := FALSE;
   BB2_RZP2.BEF_NHV.Bef.Res_23 := FALSE;
   BB2_RZP2.BEF_NHV.Bef.Res_24 := FALSE;
   BB2_RZP2.BEF_NHV.Bef.Res_25 := FALSE;
   BB2_RZP2.BEF_NHV.Bef.Res_26 := FALSE;
   BB2_RZP2.BEF_NHV.Bef.Res_27 := FALSE;
   BB2_RZP2.BEF_NHV.Bef.Res_28 := FALSE;
   BB2_RZP2.BEF_NHV.Bef.Res_29 := FALSE;
   BB2_RZP2.BEF_NHV.Bef.BF_Set_SW_chg := FALSE;
   BB2_RZP2.BEF_NHV.Bef.BF_Quit := FALSE;
   BB2_RZP2.BEF_NHV.SW_Hand := 0.0;
   BB2_UeSP.Typ := 0;
   BB2_UeSP.Idx := 18;
   BB2_UeSP.BA_VW_Hand := FALSE;
   BB2_UeSP.Tmr_VZ_Anlauf_Q := FALSE;
   BB2_UeSP.SS := FALSE;
   BB2_UeSP.SSnq := FALSE;
   BB2_UeSP.SSfq := TRUE;
   BB2_UeSP.nBB := FALSE;
   BB2_UeSP.VW_Hand_St1 := FALSE;
   BB2_UeSP.VW_Hand_St2 := FALSE;
   BB2_UeSP.VW_Hand_Stop := FALSE;
   BB2_UeSP.VW_Auto_St1 := FALSE;
   BB2_UeSP.VW_Auto_St2 := FALSE;
   BB2_UeSP.Anst_Req_St1 := FALSE;
   BB2_UeSP.Anst_Req_St2 := FALSE;
   BB2_UeSP.FM_Betrieb_Ein := FALSE;
   BB2_UeSP.FM_Betrieb_Aus := TRUE;
   BB2_UeSP.NLZ_MAZ_St1 := FALSE;
   BB2_UeSP.NLZ_MAZ_St2 := FALSE;
   BB2_UeSP.NLZ_Rev_SS_St1 := FALSE;
   BB2_UeSP.NLZ_Rev_SS_St2 := FALSE;
   BB2_UeSP.Th_St := FALSE;
   BB2_UeSP.DMA_St := FALSE;
   BB2_UeSP.DMZ_St := FALSE;
   BB2_UeSP.FU_St := FALSE;
   BB2_UeSP.TL_St := FALSE;
   BB2_UeSP.UDr_St := FALSE;
   BB2_UeSP.UeDr_St := FALSE;
   BB2_UeSP.UT_St := FALSE;
   BB2_UeSP.Le_St := FALSE;
   BB2_UeSP.UeLM_St := FALSE;
   BB2_UeSP.UeLE_St := FALSE;
   BB2_UeSP.Kom_DP_St := FALSE;
   BB2_UeSP.Kom_int_St := FALSE;
   BB2_UeSP.int_St := FALSE;
   BB2_UeSP.LZ_St := FALSE;
   BB2_UeSP.BefLZ_St := FALSE;
   BB2_UeSP.FM_GlobalQuit := FALSE;
   BB2_UeSP.Quit_RST := FALSE;
   BB2_UeSP.Tmr_VZ_Anlauf := 0;
   BB2_UeSP.Tmr_VZ_ESZ := 0;
   BB2_UeSP.Tmr_Th_St := 0;
   BB2_UeSP.Tmr_DMA_St := 0;
   BB2_UeSP.Tmr_DMZ_St := 0;
   BB2_UeSP.Tmr_FU_St := 0;
   BB2_UeSP.Tmr_TL_St := 0;
   BB2_UeSP.Tmr_UDr_St := 0;
   BB2_UeSP.Tmr_UeDr_St := 0;
   BB2_UeSP.Tmr_UT_St := 0;
   BB2_UeSP.Tmr_Le_St := 0;
   BB2_UeSP.Tmr_UeLM_St := 0;
   BB2_UeSP.Tmr_UeLE_St := 0;
   BB2_UeSP.Tmr_Kom_DP_St := 0;
   BB2_UeSP.Tmr_Kom_int_St := 0;
   BB2_UeSP.Tmr_int_St := 0;
   BB2_UeSP.Tmr_LZ_St := 0;
   BB2_UeSP.Tmr_BefLZ_St := 0;
   BB2_UeSP.Tmr_ASZ_St1 := 0;
   BB2_UeSP.Tmr_ASZ_St2 := 0;
   BB2_UeSP.Tmr_Rev_St1 := 0;
   BB2_UeSP.Tmr_Rev_St2 := 0;
   BB2_UeSP.BZ_ges_s := 375;
   BB2_UeSP.Tmr_Quit_RST := 0;
   BB2_UeSP.BEF_NHV.Bef.Bed_Res := FALSE;
   BB2_UeSP.BEF_NHV.Bef.Bed_UV := FALSE;
   BB2_UeSP.BEF_NHV.Bef.Bed_NHV := FALSE;
   BB2_UeSP.BEF_NHV.Bef.Bed_PLS := FALSE;
   BB2_UeSP.BEF_NHV.Bef.BA_Hand := FALSE;
   BB2_UeSP.BEF_NHV.Bef.BA_Auto := FALSE;
   BB2_UeSP.BEF_NHV.Bef.BF_Ein1 := FALSE;
   BB2_UeSP.BEF_NHV.Bef.BF_Ein2 := FALSE;
   BB2_UeSP.BEF_NHV.Bef.BF_Aus := FALSE;
   BB2_UeSP.BEF_NHV.Bef.BZ_Res := FALSE;
   BB2_UeSP.BEF_NHV.Bef.Res_10 := FALSE;
   BB2_UeSP.BEF_NHV.Bef.Res_11 := FALSE;
   BB2_UeSP.BEF_NHV.Bef.Res_12 := FALSE;
   BB2_UeSP.BEF_NHV.Bef.Res_13 := FALSE;
   BB2_UeSP.BEF_NHV.Bef.Res_14 := FALSE;
   BB2_UeSP.BEF_NHV.Bef.Res_15 := FALSE;
   BB2_UeSP.BEF_NHV.Bef.Res_16 := FALSE;
   BB2_UeSP.BEF_NHV.Bef.Res_17 := FALSE;
   BB2_UeSP.BEF_NHV.Bef.Res_18 := FALSE;
   BB2_UeSP.BEF_NHV.Bef.Res_19 := FALSE;
   BB2_UeSP.BEF_NHV.Bef.Res_20 := FALSE;
   BB2_UeSP.BEF_NHV.Bef.Res_21 := FALSE;
   BB2_UeSP.BEF_NHV.Bef.Res_22 := FALSE;
   BB2_UeSP.BEF_NHV.Bef.Res_23 := FALSE;
   BB2_UeSP.BEF_NHV.Bef.Res_24 := FALSE;
   BB2_UeSP.BEF_NHV.Bef.Res_25 := FALSE;
   BB2_UeSP.BEF_NHV.Bef.Res_26 := FALSE;
   BB2_UeSP.BEF_NHV.Bef.Res_27 := FALSE;
   BB2_UeSP.BEF_NHV.Bef.Res_28 := FALSE;
   BB2_UeSP.BEF_NHV.Bef.Res_29 := FALSE;
   BB2_UeSP.BEF_NHV.Bef.BF_Set_SW_chg := FALSE;
   BB2_UeSP.BEF_NHV.Bef.BF_Quit := FALSE;
   BB2_UeSP.BEF_NHV.SW_Hand := 0.0;
   BB2_AS1.Typ := 5;
   BB2_AS1.Idx := 19;
   BB2_AS1.BA_VW_Hand := FALSE;
   BB2_AS1.Tmr_VZ_Anlauf_Q := FALSE;
   BB2_AS1.SS := FALSE;
   BB2_AS1.SSnq := FALSE;
   BB2_AS1.SSfq := TRUE;
   BB2_AS1.nBB := FALSE;
   BB2_AS1.VW_Hand_St1 := FALSE;
   BB2_AS1.VW_Hand_St2 := FALSE;
   BB2_AS1.VW_Hand_Stop := FALSE;
   BB2_AS1.VW_Auto_St1 := FALSE;
   BB2_AS1.VW_Auto_St2 := FALSE;
   BB2_AS1.Anst_Req_St1 := FALSE;
   BB2_AS1.Anst_Req_St2 := FALSE;
   BB2_AS1.FM_Betrieb_Ein := FALSE;
   BB2_AS1.FM_Betrieb_Aus := TRUE;
   BB2_AS1.NLZ_MAZ_St1 := FALSE;
   BB2_AS1.NLZ_MAZ_St2 := FALSE;
   BB2_AS1.NLZ_Rev_SS_St1 := FALSE;
   BB2_AS1.NLZ_Rev_SS_St2 := FALSE;
   BB2_AS1.Th_St := FALSE;
   BB2_AS1.DMA_St := FALSE;
   BB2_AS1.DMZ_St := FALSE;
   BB2_AS1.FU_St := FALSE;
   BB2_AS1.TL_St := FALSE;
   BB2_AS1.UDr_St := FALSE;
   BB2_AS1.UeDr_St := FALSE;
   BB2_AS1.UT_St := FALSE;
   BB2_AS1.Le_St := FALSE;
   BB2_AS1.UeLM_St := FALSE;
   BB2_AS1.UeLE_St := FALSE;
   BB2_AS1.Kom_DP_St := FALSE;
   BB2_AS1.Kom_int_St := FALSE;
   BB2_AS1.int_St := FALSE;
   BB2_AS1.LZ_St := FALSE;
   BB2_AS1.BefLZ_St := FALSE;
   BB2_AS1.FM_GlobalQuit := FALSE;
   BB2_AS1.Quit_RST := FALSE;
   BB2_AS1.Tmr_VZ_Anlauf := 0;
   BB2_AS1.Tmr_VZ_ESZ := 0;
   BB2_AS1.Tmr_Th_St := 0;
   BB2_AS1.Tmr_DMA_St := 0;
   BB2_AS1.Tmr_DMZ_St := 0;
   BB2_AS1.Tmr_FU_St := 0;
   BB2_AS1.Tmr_TL_St := 0;
   BB2_AS1.Tmr_UDr_St := 0;
   BB2_AS1.Tmr_UeDr_St := 0;
   BB2_AS1.Tmr_UT_St := 0;
   BB2_AS1.Tmr_Le_St := 0;
   BB2_AS1.Tmr_UeLM_St := 0;
   BB2_AS1.Tmr_UeLE_St := 0;
   BB2_AS1.Tmr_Kom_DP_St := 0;
   BB2_AS1.Tmr_Kom_int_St := 0;
   BB2_AS1.Tmr_int_St := 0;
   BB2_AS1.Tmr_LZ_St := 0;
   BB2_AS1.Tmr_BefLZ_St := 0;
   BB2_AS1.Tmr_ASZ_St1 := 0;
   BB2_AS1.Tmr_ASZ_St2 := 0;
   BB2_AS1.Tmr_Rev_St1 := 0;
   BB2_AS1.Tmr_Rev_St2 := 0;
   BB2_AS1.BZ_ges_s := 2005;
   BB2_AS1.Tmr_Quit_RST := 0;
   BB2_AS1.BEF_NHV.Bef.Bed_Res := FALSE;
   BB2_AS1.BEF_NHV.Bef.Bed_UV := FALSE;
   BB2_AS1.BEF_NHV.Bef.Bed_NHV := FALSE;
   BB2_AS1.BEF_NHV.Bef.Bed_PLS := FALSE;
   BB2_AS1.BEF_NHV.Bef.BA_Hand := FALSE;
   BB2_AS1.BEF_NHV.Bef.BA_Auto := FALSE;
   BB2_AS1.BEF_NHV.Bef.BF_Ein1 := FALSE;
   BB2_AS1.BEF_NHV.Bef.BF_Ein2 := FALSE;
   BB2_AS1.BEF_NHV.Bef.BF_Aus := FALSE;
   BB2_AS1.BEF_NHV.Bef.BZ_Res := FALSE;
   BB2_AS1.BEF_NHV.Bef.Res_10 := FALSE;
   BB2_AS1.BEF_NHV.Bef.Res_11 := FALSE;
   BB2_AS1.BEF_NHV.Bef.Res_12 := FALSE;
   BB2_AS1.BEF_NHV.Bef.Res_13 := FALSE;
   BB2_AS1.BEF_NHV.Bef.Res_14 := FALSE;
   BB2_AS1.BEF_NHV.Bef.Res_15 := FALSE;
   BB2_AS1.BEF_NHV.Bef.Res_16 := FALSE;
   BB2_AS1.BEF_NHV.Bef.Res_17 := FALSE;
   BB2_AS1.BEF_NHV.Bef.Res_18 := FALSE;
   BB2_AS1.BEF_NHV.Bef.Res_19 := FALSE;
   BB2_AS1.BEF_NHV.Bef.Res_20 := FALSE;
   BB2_AS1.BEF_NHV.Bef.Res_21 := FALSE;
   BB2_AS1.BEF_NHV.Bef.Res_22 := FALSE;
   BB2_AS1.BEF_NHV.Bef.Res_23 := FALSE;
   BB2_AS1.BEF_NHV.Bef.Res_24 := FALSE;
   BB2_AS1.BEF_NHV.Bef.Res_25 := FALSE;
   BB2_AS1.BEF_NHV.Bef.Res_26 := FALSE;
   BB2_AS1.BEF_NHV.Bef.Res_27 := FALSE;
   BB2_AS1.BEF_NHV.Bef.Res_28 := FALSE;
   BB2_AS1.BEF_NHV.Bef.Res_29 := FALSE;
   BB2_AS1.BEF_NHV.Bef.BF_Set_SW_chg := FALSE;
   BB2_AS1.BEF_NHV.Bef.BF_Quit := FALSE;
   BB2_AS1.BEF_NHV.SW_Hand := 0.0;
   BB2_AS2.Typ := 5;
   BB2_AS2.Idx := 20;
   BB2_AS2.BA_VW_Hand := FALSE;
   BB2_AS2.Tmr_VZ_Anlauf_Q := FALSE;
   BB2_AS2.SS := FALSE;
   BB2_AS2.SSnq := FALSE;
   BB2_AS2.SSfq := TRUE;
   BB2_AS2.nBB := FALSE;
   BB2_AS2.VW_Hand_St1 := FALSE;
   BB2_AS2.VW_Hand_St2 := FALSE;
   BB2_AS2.VW_Hand_Stop := FALSE;
   BB2_AS2.VW_Auto_St1 := FALSE;
   BB2_AS2.VW_Auto_St2 := FALSE;
   BB2_AS2.Anst_Req_St1 := FALSE;
   BB2_AS2.Anst_Req_St2 := FALSE;
   BB2_AS2.FM_Betrieb_Ein := FALSE;
   BB2_AS2.FM_Betrieb_Aus := TRUE;
   BB2_AS2.NLZ_MAZ_St1 := FALSE;
   BB2_AS2.NLZ_MAZ_St2 := FALSE;
   BB2_AS2.NLZ_Rev_SS_St1 := FALSE;
   BB2_AS2.NLZ_Rev_SS_St2 := FALSE;
   BB2_AS2.Th_St := FALSE;
   BB2_AS2.DMA_St := FALSE;
   BB2_AS2.DMZ_St := FALSE;
   BB2_AS2.FU_St := FALSE;
   BB2_AS2.TL_St := FALSE;
   BB2_AS2.UDr_St := FALSE;
   BB2_AS2.UeDr_St := FALSE;
   BB2_AS2.UT_St := FALSE;
   BB2_AS2.Le_St := FALSE;
   BB2_AS2.UeLM_St := FALSE;
   BB2_AS2.UeLE_St := FALSE;
   BB2_AS2.Kom_DP_St := FALSE;
   BB2_AS2.Kom_int_St := FALSE;
   BB2_AS2.int_St := FALSE;
   BB2_AS2.LZ_St := FALSE;
   BB2_AS2.BefLZ_St := FALSE;
   BB2_AS2.FM_GlobalQuit := FALSE;
   BB2_AS2.Quit_RST := FALSE;
   BB2_AS2.Tmr_VZ_Anlauf := 0;
   BB2_AS2.Tmr_VZ_ESZ := 0;
   BB2_AS2.Tmr_Th_St := 0;
   BB2_AS2.Tmr_DMA_St := 0;
   BB2_AS2.Tmr_DMZ_St := 0;
   BB2_AS2.Tmr_FU_St := 0;
   BB2_AS2.Tmr_TL_St := 0;
   BB2_AS2.Tmr_UDr_St := 0;
   BB2_AS2.Tmr_UeDr_St := 0;
   BB2_AS2.Tmr_UT_St := 0;
   BB2_AS2.Tmr_Le_St := 0;
   BB2_AS2.Tmr_UeLM_St := 0;
   BB2_AS2.Tmr_UeLE_St := 0;
   BB2_AS2.Tmr_Kom_DP_St := 0;
   BB2_AS2.Tmr_Kom_int_St := 0;
   BB2_AS2.Tmr_int_St := 0;
   BB2_AS2.Tmr_LZ_St := 0;
   BB2_AS2.Tmr_BefLZ_St := 0;
   BB2_AS2.Tmr_ASZ_St1 := 0;
   BB2_AS2.Tmr_ASZ_St2 := 0;
   BB2_AS2.Tmr_Rev_St1 := 0;
   BB2_AS2.Tmr_Rev_St2 := 0;
   BB2_AS2.BZ_ges_s := 1909;
   BB2_AS2.Tmr_Quit_RST := 0;
   BB2_AS2.BEF_NHV.Bef.Bed_Res := FALSE;
   BB2_AS2.BEF_NHV.Bef.Bed_UV := FALSE;
   BB2_AS2.BEF_NHV.Bef.Bed_NHV := FALSE;
   BB2_AS2.BEF_NHV.Bef.Bed_PLS := FALSE;
   BB2_AS2.BEF_NHV.Bef.BA_Hand := FALSE;
   BB2_AS2.BEF_NHV.Bef.BA_Auto := FALSE;
   BB2_AS2.BEF_NHV.Bef.BF_Ein1 := FALSE;
   BB2_AS2.BEF_NHV.Bef.BF_Ein2 := FALSE;
   BB2_AS2.BEF_NHV.Bef.BF_Aus := FALSE;
   BB2_AS2.BEF_NHV.Bef.BZ_Res := FALSE;
   BB2_AS2.BEF_NHV.Bef.Res_10 := FALSE;
   BB2_AS2.BEF_NHV.Bef.Res_11 := FALSE;
   BB2_AS2.BEF_NHV.Bef.Res_12 := FALSE;
   BB2_AS2.BEF_NHV.Bef.Res_13 := FALSE;
   BB2_AS2.BEF_NHV.Bef.Res_14 := FALSE;
   BB2_AS2.BEF_NHV.Bef.Res_15 := FALSE;
   BB2_AS2.BEF_NHV.Bef.Res_16 := FALSE;
   BB2_AS2.BEF_NHV.Bef.Res_17 := FALSE;
   BB2_AS2.BEF_NHV.Bef.Res_18 := FALSE;
   BB2_AS2.BEF_NHV.Bef.Res_19 := FALSE;
   BB2_AS2.BEF_NHV.Bef.Res_20 := FALSE;
   BB2_AS2.BEF_NHV.Bef.Res_21 := FALSE;
   BB2_AS2.BEF_NHV.Bef.Res_22 := FALSE;
   BB2_AS2.BEF_NHV.Bef.Res_23 := FALSE;
   BB2_AS2.BEF_NHV.Bef.Res_24 := FALSE;
   BB2_AS2.BEF_NHV.Bef.Res_25 := FALSE;
   BB2_AS2.BEF_NHV.Bef.Res_26 := FALSE;
   BB2_AS2.BEF_NHV.Bef.Res_27 := FALSE;
   BB2_AS2.BEF_NHV.Bef.Res_28 := FALSE;
   BB2_AS2.BEF_NHV.Bef.Res_29 := FALSE;
   BB2_AS2.BEF_NHV.Bef.BF_Set_SW_chg := FALSE;
   BB2_AS2.BEF_NHV.Bef.BF_Quit := FALSE;
   BB2_AS2.BEF_NHV.SW_Hand := 0.0;
   BB2_SR1.Typ := 7;
   BB2_SR1.Idx := 21;
   BB2_SR1.BA_VW_Hand := FALSE;
   BB2_SR1.Tmr_VZ_Anlauf_Q := FALSE;
   BB2_SR1.SS := FALSE;
   BB2_SR1.SSnq := FALSE;
   BB2_SR1.SSfq := TRUE;
   BB2_SR1.nBB := FALSE;
   BB2_SR1.VW_Hand_St1 := FALSE;
   BB2_SR1.VW_Hand_St2 := FALSE;
   BB2_SR1.VW_Hand_Stop := FALSE;
   BB2_SR1.VW_Auto_St1 := FALSE;
   BB2_SR1.VW_Auto_St2 := FALSE;
   BB2_SR1.Anst_Req_St1 := FALSE;
   BB2_SR1.Anst_Req_St2 := FALSE;
   BB2_SR1.FM_Betrieb_Ein := FALSE;
   BB2_SR1.FM_Betrieb_Aus := TRUE;
   BB2_SR1.NLZ_MAZ_St1 := FALSE;
   BB2_SR1.NLZ_MAZ_St2 := FALSE;
   BB2_SR1.NLZ_Rev_SS_St1 := FALSE;
   BB2_SR1.NLZ_Rev_SS_St2 := FALSE;
   BB2_SR1.Th_St := FALSE;
   BB2_SR1.DMA_St := FALSE;
   BB2_SR1.DMZ_St := FALSE;
   BB2_SR1.FU_St := FALSE;
   BB2_SR1.TL_St := FALSE;
   BB2_SR1.UDr_St := FALSE;
   BB2_SR1.UeDr_St := FALSE;
   BB2_SR1.UT_St := FALSE;
   BB2_SR1.Le_St := FALSE;
   BB2_SR1.UeLM_St := FALSE;
   BB2_SR1.UeLE_St := FALSE;
   BB2_SR1.Kom_DP_St := FALSE;
   BB2_SR1.Kom_int_St := FALSE;
   BB2_SR1.int_St := FALSE;
   BB2_SR1.LZ_St := FALSE;
   BB2_SR1.BefLZ_St := FALSE;
   BB2_SR1.FM_GlobalQuit := FALSE;
   BB2_SR1.Quit_RST := FALSE;
   BB2_SR1.Tmr_VZ_Anlauf := 0;
   BB2_SR1.Tmr_VZ_ESZ := 0;
   BB2_SR1.Tmr_Th_St := 0;
   BB2_SR1.Tmr_DMA_St := 0;
   BB2_SR1.Tmr_DMZ_St := 0;
   BB2_SR1.Tmr_FU_St := 0;
   BB2_SR1.Tmr_TL_St := 0;
   BB2_SR1.Tmr_UDr_St := 0;
   BB2_SR1.Tmr_UeDr_St := 0;
   BB2_SR1.Tmr_UT_St := 0;
   BB2_SR1.Tmr_Le_St := 0;
   BB2_SR1.Tmr_UeLM_St := 0;
   BB2_SR1.Tmr_UeLE_St := 0;
   BB2_SR1.Tmr_Kom_DP_St := 0;
   BB2_SR1.Tmr_Kom_int_St := 0;
   BB2_SR1.Tmr_int_St := 0;
   BB2_SR1.Tmr_LZ_St := 0;
   BB2_SR1.Tmr_BefLZ_St := 0;
   BB2_SR1.Tmr_ASZ_St1 := 0;
   BB2_SR1.Tmr_ASZ_St2 := 0;
   BB2_SR1.Tmr_Rev_St1 := 0;
   BB2_SR1.Tmr_Rev_St2 := 0;
   BB2_SR1.BZ_ges_s := 2516;
   BB2_SR1.Tmr_Quit_RST := 0;
   BB2_SR1.BEF_NHV.Bef.Bed_Res := FALSE;
   BB2_SR1.BEF_NHV.Bef.Bed_UV := FALSE;
   BB2_SR1.BEF_NHV.Bef.Bed_NHV := FALSE;
   BB2_SR1.BEF_NHV.Bef.Bed_PLS := FALSE;
   BB2_SR1.BEF_NHV.Bef.BA_Hand := FALSE;
   BB2_SR1.BEF_NHV.Bef.BA_Auto := FALSE;
   BB2_SR1.BEF_NHV.Bef.BF_Ein1 := FALSE;
   BB2_SR1.BEF_NHV.Bef.BF_Ein2 := FALSE;
   BB2_SR1.BEF_NHV.Bef.BF_Aus := FALSE;
   BB2_SR1.BEF_NHV.Bef.BZ_Res := FALSE;
   BB2_SR1.BEF_NHV.Bef.Res_10 := FALSE;
   BB2_SR1.BEF_NHV.Bef.Res_11 := FALSE;
   BB2_SR1.BEF_NHV.Bef.Res_12 := FALSE;
   BB2_SR1.BEF_NHV.Bef.Res_13 := FALSE;
   BB2_SR1.BEF_NHV.Bef.Res_14 := FALSE;
   BB2_SR1.BEF_NHV.Bef.Res_15 := FALSE;
   BB2_SR1.BEF_NHV.Bef.Res_16 := FALSE;
   BB2_SR1.BEF_NHV.Bef.Res_17 := FALSE;
   BB2_SR1.BEF_NHV.Bef.Res_18 := FALSE;
   BB2_SR1.BEF_NHV.Bef.Res_19 := FALSE;
   BB2_SR1.BEF_NHV.Bef.Res_20 := FALSE;
   BB2_SR1.BEF_NHV.Bef.Res_21 := FALSE;
   BB2_SR1.BEF_NHV.Bef.Res_22 := FALSE;
   BB2_SR1.BEF_NHV.Bef.Res_23 := FALSE;
   BB2_SR1.BEF_NHV.Bef.Res_24 := FALSE;
   BB2_SR1.BEF_NHV.Bef.Res_25 := FALSE;
   BB2_SR1.BEF_NHV.Bef.Res_26 := FALSE;
   BB2_SR1.BEF_NHV.Bef.Res_27 := FALSE;
   BB2_SR1.BEF_NHV.Bef.Res_28 := FALSE;
   BB2_SR1.BEF_NHV.Bef.Res_29 := FALSE;
   BB2_SR1.BEF_NHV.Bef.BF_Set_SW_chg := FALSE;
   BB2_SR1.BEF_NHV.Bef.BF_Quit := FALSE;
   BB2_SR1.BEF_NHV.SW_Hand := 0.0;
   BB2_SR2.Typ := 7;
   BB2_SR2.Idx := 22;
   BB2_SR2.BA_VW_Hand := FALSE;
   BB2_SR2.Tmr_VZ_Anlauf_Q := FALSE;
   BB2_SR2.SS := FALSE;
   BB2_SR2.SSnq := FALSE;
   BB2_SR2.SSfq := TRUE;
   BB2_SR2.nBB := FALSE;
   BB2_SR2.VW_Hand_St1 := FALSE;
   BB2_SR2.VW_Hand_St2 := FALSE;
   BB2_SR2.VW_Hand_Stop := FALSE;
   BB2_SR2.VW_Auto_St1 := FALSE;
   BB2_SR2.VW_Auto_St2 := FALSE;
   BB2_SR2.Anst_Req_St1 := FALSE;
   BB2_SR2.Anst_Req_St2 := FALSE;
   BB2_SR2.FM_Betrieb_Ein := FALSE;
   BB2_SR2.FM_Betrieb_Aus := TRUE;
   BB2_SR2.NLZ_MAZ_St1 := FALSE;
   BB2_SR2.NLZ_MAZ_St2 := FALSE;
   BB2_SR2.NLZ_Rev_SS_St1 := FALSE;
   BB2_SR2.NLZ_Rev_SS_St2 := FALSE;
   BB2_SR2.Th_St := FALSE;
   BB2_SR2.DMA_St := FALSE;
   BB2_SR2.DMZ_St := FALSE;
   BB2_SR2.FU_St := FALSE;
   BB2_SR2.TL_St := FALSE;
   BB2_SR2.UDr_St := FALSE;
   BB2_SR2.UeDr_St := FALSE;
   BB2_SR2.UT_St := FALSE;
   BB2_SR2.Le_St := FALSE;
   BB2_SR2.UeLM_St := FALSE;
   BB2_SR2.UeLE_St := FALSE;
   BB2_SR2.Kom_DP_St := FALSE;
   BB2_SR2.Kom_int_St := FALSE;
   BB2_SR2.int_St := FALSE;
   BB2_SR2.LZ_St := FALSE;
   BB2_SR2.BefLZ_St := FALSE;
   BB2_SR2.FM_GlobalQuit := FALSE;
   BB2_SR2.Quit_RST := FALSE;
   BB2_SR2.Tmr_VZ_Anlauf := 0;
   BB2_SR2.Tmr_VZ_ESZ := 0;
   BB2_SR2.Tmr_Th_St := 0;
   BB2_SR2.Tmr_DMA_St := 0;
   BB2_SR2.Tmr_DMZ_St := 0;
   BB2_SR2.Tmr_FU_St := 0;
   BB2_SR2.Tmr_TL_St := 0;
   BB2_SR2.Tmr_UDr_St := 0;
   BB2_SR2.Tmr_UeDr_St := 0;
   BB2_SR2.Tmr_UT_St := 0;
   BB2_SR2.Tmr_Le_St := 0;
   BB2_SR2.Tmr_UeLM_St := 0;
   BB2_SR2.Tmr_UeLE_St := 0;
   BB2_SR2.Tmr_Kom_DP_St := 0;
   BB2_SR2.Tmr_Kom_int_St := 0;
   BB2_SR2.Tmr_int_St := 0;
   BB2_SR2.Tmr_LZ_St := 0;
   BB2_SR2.Tmr_BefLZ_St := 0;
   BB2_SR2.Tmr_ASZ_St1 := 0;
   BB2_SR2.Tmr_ASZ_St2 := 0;
   BB2_SR2.Tmr_Rev_St1 := 0;
   BB2_SR2.Tmr_Rev_St2 := 0;
   BB2_SR2.BZ_ges_s := 2516;
   BB2_SR2.Tmr_Quit_RST := 0;
   BB2_SR2.BEF_NHV.Bef.Bed_Res := FALSE;
   BB2_SR2.BEF_NHV.Bef.Bed_UV := FALSE;
   BB2_SR2.BEF_NHV.Bef.Bed_NHV := FALSE;
   BB2_SR2.BEF_NHV.Bef.Bed_PLS := FALSE;
   BB2_SR2.BEF_NHV.Bef.BA_Hand := FALSE;
   BB2_SR2.BEF_NHV.Bef.BA_Auto := FALSE;
   BB2_SR2.BEF_NHV.Bef.BF_Ein1 := FALSE;
   BB2_SR2.BEF_NHV.Bef.BF_Ein2 := FALSE;
   BB2_SR2.BEF_NHV.Bef.BF_Aus := FALSE;
   BB2_SR2.BEF_NHV.Bef.BZ_Res := FALSE;
   BB2_SR2.BEF_NHV.Bef.Res_10 := FALSE;
   BB2_SR2.BEF_NHV.Bef.Res_11 := FALSE;
   BB2_SR2.BEF_NHV.Bef.Res_12 := FALSE;
   BB2_SR2.BEF_NHV.Bef.Res_13 := FALSE;
   BB2_SR2.BEF_NHV.Bef.Res_14 := FALSE;
   BB2_SR2.BEF_NHV.Bef.Res_15 := FALSE;
   BB2_SR2.BEF_NHV.Bef.Res_16 := FALSE;
   BB2_SR2.BEF_NHV.Bef.Res_17 := FALSE;
   BB2_SR2.BEF_NHV.Bef.Res_18 := FALSE;
   BB2_SR2.BEF_NHV.Bef.Res_19 := FALSE;
   BB2_SR2.BEF_NHV.Bef.Res_20 := FALSE;
   BB2_SR2.BEF_NHV.Bef.Res_21 := FALSE;
   BB2_SR2.BEF_NHV.Bef.Res_22 := FALSE;
   BB2_SR2.BEF_NHV.Bef.Res_23 := FALSE;
   BB2_SR2.BEF_NHV.Bef.Res_24 := FALSE;
   BB2_SR2.BEF_NHV.Bef.Res_25 := FALSE;
   BB2_SR2.BEF_NHV.Bef.Res_26 := FALSE;
   BB2_SR2.BEF_NHV.Bef.Res_27 := FALSE;
   BB2_SR2.BEF_NHV.Bef.Res_28 := FALSE;
   BB2_SR2.BEF_NHV.Bef.Res_29 := FALSE;
   BB2_SR2.BEF_NHV.Bef.BF_Set_SW_chg := FALSE;
   BB2_SR2.BEF_NHV.Bef.BF_Quit := FALSE;
   BB2_SR2.BEF_NHV.SW_Hand := 0.0;
   BB1_SR_K.Typ := 0;
   BB1_SR_K.Idx := 23;
   BB1_SR_K.BA_VW_Hand := FALSE;
   BB1_SR_K.Tmr_VZ_Anlauf_Q := TRUE;
   BB1_SR_K.SS := TRUE;
   BB1_SR_K.SSnq := FALSE;
   BB1_SR_K.SSfq := FALSE;
   BB1_SR_K.nBB := TRUE;
   BB1_SR_K.VW_Hand_St1 := FALSE;
   BB1_SR_K.VW_Hand_St2 := FALSE;
   BB1_SR_K.VW_Hand_Stop := FALSE;
   BB1_SR_K.VW_Auto_St1 := FALSE;
   BB1_SR_K.VW_Auto_St2 := FALSE;
   BB1_SR_K.Anst_Req_St1 := FALSE;
   BB1_SR_K.Anst_Req_St2 := FALSE;
   BB1_SR_K.FM_Betrieb_Ein := TRUE;
   BB1_SR_K.FM_Betrieb_Aus := FALSE;
   BB1_SR_K.NLZ_MAZ_St1 := FALSE;
   BB1_SR_K.NLZ_MAZ_St2 := FALSE;
   BB1_SR_K.NLZ_Rev_SS_St1 := FALSE;
   BB1_SR_K.NLZ_Rev_SS_St2 := FALSE;
   BB1_SR_K.Th_St := TRUE;
   BB1_SR_K.DMA_St := FALSE;
   BB1_SR_K.DMZ_St := FALSE;
   BB1_SR_K.FU_St := FALSE;
   BB1_SR_K.TL_St := FALSE;
   BB1_SR_K.UDr_St := FALSE;
   BB1_SR_K.UeDr_St := FALSE;
   BB1_SR_K.UT_St := FALSE;
   BB1_SR_K.Le_St := FALSE;
   BB1_SR_K.UeLM_St := FALSE;
   BB1_SR_K.UeLE_St := FALSE;
   BB1_SR_K.Kom_DP_St := FALSE;
   BB1_SR_K.Kom_int_St := FALSE;
   BB1_SR_K.int_St := FALSE;
   BB1_SR_K.LZ_St := FALSE;
   BB1_SR_K.BefLZ_St := FALSE;
   BB1_SR_K.FM_GlobalQuit := FALSE;
   BB1_SR_K.Quit_RST := FALSE;
   BB1_SR_K.Tmr_VZ_Anlauf := 3;
   BB1_SR_K.Tmr_VZ_ESZ := 0;
   BB1_SR_K.Tmr_Th_St := 5;
   BB1_SR_K.Tmr_DMA_St := 0;
   BB1_SR_K.Tmr_DMZ_St := 0;
   BB1_SR_K.Tmr_FU_St := 0;
   BB1_SR_K.Tmr_TL_St := 0;
   BB1_SR_K.Tmr_UDr_St := 0;
   BB1_SR_K.Tmr_UeDr_St := 0;
   BB1_SR_K.Tmr_UT_St := 0;
   BB1_SR_K.Tmr_Le_St := 0;
   BB1_SR_K.Tmr_UeLM_St := 0;
   BB1_SR_K.Tmr_UeLE_St := 0;
   BB1_SR_K.Tmr_Kom_DP_St := 0;
   BB1_SR_K.Tmr_Kom_int_St := 0;
   BB1_SR_K.Tmr_int_St := 0;
   BB1_SR_K.Tmr_LZ_St := 0;
   BB1_SR_K.Tmr_BefLZ_St := 0;
   BB1_SR_K.Tmr_ASZ_St1 := 0;
   BB1_SR_K.Tmr_ASZ_St2 := 0;
   BB1_SR_K.Tmr_Rev_St1 := 0;
   BB1_SR_K.Tmr_Rev_St2 := 0;
   BB1_SR_K.BZ_ges_s := 2529;
   BB1_SR_K.Tmr_Quit_RST := 0;
   BB1_SR_K.BEF_NHV.Bef.Bed_Res := FALSE;
   BB1_SR_K.BEF_NHV.Bef.Bed_UV := FALSE;
   BB1_SR_K.BEF_NHV.Bef.Bed_NHV := FALSE;
   BB1_SR_K.BEF_NHV.Bef.Bed_PLS := FALSE;
   BB1_SR_K.BEF_NHV.Bef.BA_Hand := FALSE;
   BB1_SR_K.BEF_NHV.Bef.BA_Auto := FALSE;
   BB1_SR_K.BEF_NHV.Bef.BF_Ein1 := FALSE;
   BB1_SR_K.BEF_NHV.Bef.BF_Ein2 := FALSE;
   BB1_SR_K.BEF_NHV.Bef.BF_Aus := FALSE;
   BB1_SR_K.BEF_NHV.Bef.BZ_Res := FALSE;
   BB1_SR_K.BEF_NHV.Bef.Res_10 := FALSE;
   BB1_SR_K.BEF_NHV.Bef.Res_11 := FALSE;
   BB1_SR_K.BEF_NHV.Bef.Res_12 := FALSE;
   BB1_SR_K.BEF_NHV.Bef.Res_13 := FALSE;
   BB1_SR_K.BEF_NHV.Bef.Res_14 := FALSE;
   BB1_SR_K.BEF_NHV.Bef.Res_15 := FALSE;
   BB1_SR_K.BEF_NHV.Bef.Res_16 := FALSE;
   BB1_SR_K.BEF_NHV.Bef.Res_17 := FALSE;
   BB1_SR_K.BEF_NHV.Bef.Res_18 := FALSE;
   BB1_SR_K.BEF_NHV.Bef.Res_19 := FALSE;
   BB1_SR_K.BEF_NHV.Bef.Res_20 := FALSE;
   BB1_SR_K.BEF_NHV.Bef.Res_21 := FALSE;
   BB1_SR_K.BEF_NHV.Bef.Res_22 := FALSE;
   BB1_SR_K.BEF_NHV.Bef.Res_23 := FALSE;
   BB1_SR_K.BEF_NHV.Bef.Res_24 := FALSE;
   BB1_SR_K.BEF_NHV.Bef.Res_25 := FALSE;
   BB1_SR_K.BEF_NHV.Bef.Res_26 := FALSE;
   BB1_SR_K.BEF_NHV.Bef.Res_27 := FALSE;
   BB1_SR_K.BEF_NHV.Bef.Res_28 := FALSE;
   BB1_SR_K.BEF_NHV.Bef.Res_29 := FALSE;
   BB1_SR_K.BEF_NHV.Bef.BF_Set_SW_chg := FALSE;
   BB1_SR_K.BEF_NHV.Bef.BF_Quit := FALSE;
   BB1_SR_K.BEF_NHV.SW_Hand := 0.0;
   Zulauf_AR_P1.Typ := 0;
   Zulauf_AR_P1.Idx := 24;
   Zulauf_AR_P1.BA_VW_Hand := FALSE;
   Zulauf_AR_P1.Tmr_VZ_Anlauf_Q := FALSE;
   Zulauf_AR_P1.SS := FALSE;
   Zulauf_AR_P1.SSnq := FALSE;
   Zulauf_AR_P1.SSfq := TRUE;
   Zulauf_AR_P1.nBB := FALSE;
   Zulauf_AR_P1.VW_Hand_St1 := FALSE;
   Zulauf_AR_P1.VW_Hand_St2 := FALSE;
   Zulauf_AR_P1.VW_Hand_Stop := FALSE;
   Zulauf_AR_P1.VW_Auto_St1 := FALSE;
   Zulauf_AR_P1.VW_Auto_St2 := FALSE;
   Zulauf_AR_P1.Anst_Req_St1 := FALSE;
   Zulauf_AR_P1.Anst_Req_St2 := FALSE;
   Zulauf_AR_P1.FM_Betrieb_Ein := FALSE;
   Zulauf_AR_P1.FM_Betrieb_Aus := TRUE;
   Zulauf_AR_P1.NLZ_MAZ_St1 := FALSE;
   Zulauf_AR_P1.NLZ_MAZ_St2 := FALSE;
   Zulauf_AR_P1.NLZ_Rev_SS_St1 := FALSE;
   Zulauf_AR_P1.NLZ_Rev_SS_St2 := FALSE;
   Zulauf_AR_P1.Th_St := FALSE;
   Zulauf_AR_P1.DMA_St := FALSE;
   Zulauf_AR_P1.DMZ_St := FALSE;
   Zulauf_AR_P1.FU_St := FALSE;
   Zulauf_AR_P1.TL_St := FALSE;
   Zulauf_AR_P1.UDr_St := FALSE;
   Zulauf_AR_P1.UeDr_St := FALSE;
   Zulauf_AR_P1.UT_St := FALSE;
   Zulauf_AR_P1.Le_St := FALSE;
   Zulauf_AR_P1.UeLM_St := FALSE;
   Zulauf_AR_P1.UeLE_St := FALSE;
   Zulauf_AR_P1.Kom_DP_St := FALSE;
   Zulauf_AR_P1.Kom_int_St := FALSE;
   Zulauf_AR_P1.int_St := FALSE;
   Zulauf_AR_P1.LZ_St := FALSE;
   Zulauf_AR_P1.BefLZ_St := FALSE;
   Zulauf_AR_P1.FM_GlobalQuit := FALSE;
   Zulauf_AR_P1.Quit_RST := FALSE;
   Zulauf_AR_P1.Tmr_VZ_Anlauf := 0;
   Zulauf_AR_P1.Tmr_VZ_ESZ := 0;
   Zulauf_AR_P1.Tmr_Th_St := 0;
   Zulauf_AR_P1.Tmr_DMA_St := 0;
   Zulauf_AR_P1.Tmr_DMZ_St := 0;
   Zulauf_AR_P1.Tmr_FU_St := 0;
   Zulauf_AR_P1.Tmr_TL_St := 0;
   Zulauf_AR_P1.Tmr_UDr_St := 0;
   Zulauf_AR_P1.Tmr_UeDr_St := 0;
   Zulauf_AR_P1.Tmr_UT_St := 0;
   Zulauf_AR_P1.Tmr_Le_St := 0;
   Zulauf_AR_P1.Tmr_UeLM_St := 0;
   Zulauf_AR_P1.Tmr_UeLE_St := 0;
   Zulauf_AR_P1.Tmr_Kom_DP_St := 0;
   Zulauf_AR_P1.Tmr_Kom_int_St := 0;
   Zulauf_AR_P1.Tmr_int_St := 0;
   Zulauf_AR_P1.Tmr_LZ_St := 0;
   Zulauf_AR_P1.Tmr_BefLZ_St := 0;
   Zulauf_AR_P1.Tmr_ASZ_St1 := 0;
   Zulauf_AR_P1.Tmr_ASZ_St2 := 0;
   Zulauf_AR_P1.Tmr_Rev_St1 := 0;
   Zulauf_AR_P1.Tmr_Rev_St2 := 0;
   Zulauf_AR_P1.BZ_ges_s := 0;
   Zulauf_AR_P1.Tmr_Quit_RST := 0;
   Zulauf_AR_P1.BEF_NHV.Bef.Bed_Res := FALSE;
   Zulauf_AR_P1.BEF_NHV.Bef.Bed_UV := FALSE;
   Zulauf_AR_P1.BEF_NHV.Bef.Bed_NHV := FALSE;
   Zulauf_AR_P1.BEF_NHV.Bef.Bed_PLS := FALSE;
   Zulauf_AR_P1.BEF_NHV.Bef.BA_Hand := FALSE;
   Zulauf_AR_P1.BEF_NHV.Bef.BA_Auto := FALSE;
   Zulauf_AR_P1.BEF_NHV.Bef.BF_Ein1 := FALSE;
   Zulauf_AR_P1.BEF_NHV.Bef.BF_Ein2 := FALSE;
   Zulauf_AR_P1.BEF_NHV.Bef.BF_Aus := FALSE;
   Zulauf_AR_P1.BEF_NHV.Bef.BZ_Res := FALSE;
   Zulauf_AR_P1.BEF_NHV.Bef.Res_10 := FALSE;
   Zulauf_AR_P1.BEF_NHV.Bef.Res_11 := FALSE;
   Zulauf_AR_P1.BEF_NHV.Bef.Res_12 := FALSE;
   Zulauf_AR_P1.BEF_NHV.Bef.Res_13 := FALSE;
   Zulauf_AR_P1.BEF_NHV.Bef.Res_14 := FALSE;
   Zulauf_AR_P1.BEF_NHV.Bef.Res_15 := FALSE;
   Zulauf_AR_P1.BEF_NHV.Bef.Res_16 := FALSE;
   Zulauf_AR_P1.BEF_NHV.Bef.Res_17 := FALSE;
   Zulauf_AR_P1.BEF_NHV.Bef.Res_18 := FALSE;
   Zulauf_AR_P1.BEF_NHV.Bef.Res_19 := FALSE;
   Zulauf_AR_P1.BEF_NHV.Bef.Res_20 := FALSE;
   Zulauf_AR_P1.BEF_NHV.Bef.Res_21 := FALSE;
   Zulauf_AR_P1.BEF_NHV.Bef.Res_22 := FALSE;
   Zulauf_AR_P1.BEF_NHV.Bef.Res_23 := FALSE;
   Zulauf_AR_P1.BEF_NHV.Bef.Res_24 := FALSE;
   Zulauf_AR_P1.BEF_NHV.Bef.Res_25 := FALSE;
   Zulauf_AR_P1.BEF_NHV.Bef.Res_26 := FALSE;
   Zulauf_AR_P1.BEF_NHV.Bef.Res_27 := FALSE;
   Zulauf_AR_P1.BEF_NHV.Bef.Res_28 := FALSE;
   Zulauf_AR_P1.BEF_NHV.Bef.Res_29 := FALSE;
   Zulauf_AR_P1.BEF_NHV.Bef.BF_Set_SW_chg := FALSE;
   Zulauf_AR_P1.BEF_NHV.Bef.BF_Quit := FALSE;
   Zulauf_AR_P1.BEF_NHV.SW_Hand := 0.0;
   Zulauf_AR_P2.Typ := 0;
   Zulauf_AR_P2.Idx := 25;
   Zulauf_AR_P2.BA_VW_Hand := FALSE;
   Zulauf_AR_P2.Tmr_VZ_Anlauf_Q := FALSE;
   Zulauf_AR_P2.SS := FALSE;
   Zulauf_AR_P2.SSnq := FALSE;
   Zulauf_AR_P2.SSfq := TRUE;
   Zulauf_AR_P2.nBB := FALSE;
   Zulauf_AR_P2.VW_Hand_St1 := FALSE;
   Zulauf_AR_P2.VW_Hand_St2 := FALSE;
   Zulauf_AR_P2.VW_Hand_Stop := FALSE;
   Zulauf_AR_P2.VW_Auto_St1 := FALSE;
   Zulauf_AR_P2.VW_Auto_St2 := FALSE;
   Zulauf_AR_P2.Anst_Req_St1 := FALSE;
   Zulauf_AR_P2.Anst_Req_St2 := FALSE;
   Zulauf_AR_P2.FM_Betrieb_Ein := FALSE;
   Zulauf_AR_P2.FM_Betrieb_Aus := TRUE;
   Zulauf_AR_P2.NLZ_MAZ_St1 := FALSE;
   Zulauf_AR_P2.NLZ_MAZ_St2 := FALSE;
   Zulauf_AR_P2.NLZ_Rev_SS_St1 := FALSE;
   Zulauf_AR_P2.NLZ_Rev_SS_St2 := FALSE;
   Zulauf_AR_P2.Th_St := FALSE;
   Zulauf_AR_P2.DMA_St := FALSE;
   Zulauf_AR_P2.DMZ_St := FALSE;
   Zulauf_AR_P2.FU_St := FALSE;
   Zulauf_AR_P2.TL_St := FALSE;
   Zulauf_AR_P2.UDr_St := FALSE;
   Zulauf_AR_P2.UeDr_St := FALSE;
   Zulauf_AR_P2.UT_St := FALSE;
   Zulauf_AR_P2.Le_St := FALSE;
   Zulauf_AR_P2.UeLM_St := FALSE;
   Zulauf_AR_P2.UeLE_St := FALSE;
   Zulauf_AR_P2.Kom_DP_St := FALSE;
   Zulauf_AR_P2.Kom_int_St := FALSE;
   Zulauf_AR_P2.int_St := FALSE;
   Zulauf_AR_P2.LZ_St := FALSE;
   Zulauf_AR_P2.BefLZ_St := FALSE;
   Zulauf_AR_P2.FM_GlobalQuit := FALSE;
   Zulauf_AR_P2.Quit_RST := FALSE;
   Zulauf_AR_P2.Tmr_VZ_Anlauf := 0;
   Zulauf_AR_P2.Tmr_VZ_ESZ := 0;
   Zulauf_AR_P2.Tmr_Th_St := 0;
   Zulauf_AR_P2.Tmr_DMA_St := 0;
   Zulauf_AR_P2.Tmr_DMZ_St := 0;
   Zulauf_AR_P2.Tmr_FU_St := 0;
   Zulauf_AR_P2.Tmr_TL_St := 0;
   Zulauf_AR_P2.Tmr_UDr_St := 0;
   Zulauf_AR_P2.Tmr_UeDr_St := 0;
   Zulauf_AR_P2.Tmr_UT_St := 0;
   Zulauf_AR_P2.Tmr_Le_St := 0;
   Zulauf_AR_P2.Tmr_UeLM_St := 0;
   Zulauf_AR_P2.Tmr_UeLE_St := 0;
   Zulauf_AR_P2.Tmr_Kom_DP_St := 0;
   Zulauf_AR_P2.Tmr_Kom_int_St := 0;
   Zulauf_AR_P2.Tmr_int_St := 0;
   Zulauf_AR_P2.Tmr_LZ_St := 0;
   Zulauf_AR_P2.Tmr_BefLZ_St := 0;
   Zulauf_AR_P2.Tmr_ASZ_St1 := 0;
   Zulauf_AR_P2.Tmr_ASZ_St2 := 0;
   Zulauf_AR_P2.Tmr_Rev_St1 := 0;
   Zulauf_AR_P2.Tmr_Rev_St2 := 0;
   Zulauf_AR_P2.BZ_ges_s := 676;
   Zulauf_AR_P2.Tmr_Quit_RST := 0;
   Zulauf_AR_P2.BEF_NHV.Bef.Bed_Res := FALSE;
   Zulauf_AR_P2.BEF_NHV.Bef.Bed_UV := FALSE;
   Zulauf_AR_P2.BEF_NHV.Bef.Bed_NHV := FALSE;
   Zulauf_AR_P2.BEF_NHV.Bef.Bed_PLS := FALSE;
   Zulauf_AR_P2.BEF_NHV.Bef.BA_Hand := FALSE;
   Zulauf_AR_P2.BEF_NHV.Bef.BA_Auto := FALSE;
   Zulauf_AR_P2.BEF_NHV.Bef.BF_Ein1 := FALSE;
   Zulauf_AR_P2.BEF_NHV.Bef.BF_Ein2 := FALSE;
   Zulauf_AR_P2.BEF_NHV.Bef.BF_Aus := FALSE;
   Zulauf_AR_P2.BEF_NHV.Bef.BZ_Res := FALSE;
   Zulauf_AR_P2.BEF_NHV.Bef.Res_10 := FALSE;
   Zulauf_AR_P2.BEF_NHV.Bef.Res_11 := FALSE;
   Zulauf_AR_P2.BEF_NHV.Bef.Res_12 := FALSE;
   Zulauf_AR_P2.BEF_NHV.Bef.Res_13 := FALSE;
   Zulauf_AR_P2.BEF_NHV.Bef.Res_14 := FALSE;
   Zulauf_AR_P2.BEF_NHV.Bef.Res_15 := FALSE;
   Zulauf_AR_P2.BEF_NHV.Bef.Res_16 := FALSE;
   Zulauf_AR_P2.BEF_NHV.Bef.Res_17 := FALSE;
   Zulauf_AR_P2.BEF_NHV.Bef.Res_18 := FALSE;
   Zulauf_AR_P2.BEF_NHV.Bef.Res_19 := FALSE;
   Zulauf_AR_P2.BEF_NHV.Bef.Res_20 := FALSE;
   Zulauf_AR_P2.BEF_NHV.Bef.Res_21 := FALSE;
   Zulauf_AR_P2.BEF_NHV.Bef.Res_22 := FALSE;
   Zulauf_AR_P2.BEF_NHV.Bef.Res_23 := FALSE;
   Zulauf_AR_P2.BEF_NHV.Bef.Res_24 := FALSE;
   Zulauf_AR_P2.BEF_NHV.Bef.Res_25 := FALSE;
   Zulauf_AR_P2.BEF_NHV.Bef.Res_26 := FALSE;
   Zulauf_AR_P2.BEF_NHV.Bef.Res_27 := FALSE;
   Zulauf_AR_P2.BEF_NHV.Bef.Res_28 := FALSE;
   Zulauf_AR_P2.BEF_NHV.Bef.Res_29 := FALSE;
   Zulauf_AR_P2.BEF_NHV.Bef.BF_Set_SW_chg := FALSE;
   Zulauf_AR_P2.BEF_NHV.Bef.BF_Quit := FALSE;
   Zulauf_AR_P2.BEF_NHV.SW_Hand := 0.0;
   Zulauf_AS.Typ := 5;
   Zulauf_AS.Idx := 26;
   Zulauf_AS.BA_VW_Hand := FALSE;
   Zulauf_AS.Tmr_VZ_Anlauf_Q := FALSE;
   Zulauf_AS.SS := FALSE;
   Zulauf_AS.SSnq := FALSE;
   Zulauf_AS.SSfq := TRUE;
   Zulauf_AS.nBB := FALSE;
   Zulauf_AS.VW_Hand_St1 := FALSE;
   Zulauf_AS.VW_Hand_St2 := FALSE;
   Zulauf_AS.VW_Hand_Stop := FALSE;
   Zulauf_AS.VW_Auto_St1 := FALSE;
   Zulauf_AS.VW_Auto_St2 := FALSE;
   Zulauf_AS.Anst_Req_St1 := FALSE;
   Zulauf_AS.Anst_Req_St2 := FALSE;
   Zulauf_AS.FM_Betrieb_Ein := FALSE;
   Zulauf_AS.FM_Betrieb_Aus := TRUE;
   Zulauf_AS.NLZ_MAZ_St1 := FALSE;
   Zulauf_AS.NLZ_MAZ_St2 := FALSE;
   Zulauf_AS.NLZ_Rev_SS_St1 := FALSE;
   Zulauf_AS.NLZ_Rev_SS_St2 := FALSE;
   Zulauf_AS.Th_St := FALSE;
   Zulauf_AS.DMA_St := FALSE;
   Zulauf_AS.DMZ_St := FALSE;
   Zulauf_AS.FU_St := FALSE;
   Zulauf_AS.TL_St := FALSE;
   Zulauf_AS.UDr_St := FALSE;
   Zulauf_AS.UeDr_St := FALSE;
   Zulauf_AS.UT_St := FALSE;
   Zulauf_AS.Le_St := FALSE;
   Zulauf_AS.UeLM_St := FALSE;
   Zulauf_AS.UeLE_St := FALSE;
   Zulauf_AS.Kom_DP_St := FALSE;
   Zulauf_AS.Kom_int_St := FALSE;
   Zulauf_AS.int_St := FALSE;
   Zulauf_AS.LZ_St := FALSE;
   Zulauf_AS.BefLZ_St := FALSE;
   Zulauf_AS.FM_GlobalQuit := FALSE;
   Zulauf_AS.Quit_RST := FALSE;
   Zulauf_AS.Tmr_VZ_Anlauf := 0;
   Zulauf_AS.Tmr_VZ_ESZ := 0;
   Zulauf_AS.Tmr_Th_St := 0;
   Zulauf_AS.Tmr_DMA_St := 0;
   Zulauf_AS.Tmr_DMZ_St := 0;
   Zulauf_AS.Tmr_FU_St := 0;
   Zulauf_AS.Tmr_TL_St := 0;
   Zulauf_AS.Tmr_UDr_St := 0;
   Zulauf_AS.Tmr_UeDr_St := 0;
   Zulauf_AS.Tmr_UT_St := 0;
   Zulauf_AS.Tmr_Le_St := 0;
   Zulauf_AS.Tmr_UeLM_St := 0;
   Zulauf_AS.Tmr_UeLE_St := 0;
   Zulauf_AS.Tmr_Kom_DP_St := 0;
   Zulauf_AS.Tmr_Kom_int_St := 0;
   Zulauf_AS.Tmr_int_St := 0;
   Zulauf_AS.Tmr_LZ_St := 0;
   Zulauf_AS.Tmr_BefLZ_St := 0;
   Zulauf_AS.Tmr_ASZ_St1 := 0;
   Zulauf_AS.Tmr_ASZ_St2 := 0;
   Zulauf_AS.Tmr_Rev_St1 := 0;
   Zulauf_AS.Tmr_Rev_St2 := 0;
   Zulauf_AS.BZ_ges_s := 0;
   Zulauf_AS.Tmr_Quit_RST := 0;
   Zulauf_AS.BEF_NHV.Bef.Bed_Res := FALSE;
   Zulauf_AS.BEF_NHV.Bef.Bed_UV := FALSE;
   Zulauf_AS.BEF_NHV.Bef.Bed_NHV := FALSE;
   Zulauf_AS.BEF_NHV.Bef.Bed_PLS := FALSE;
   Zulauf_AS.BEF_NHV.Bef.BA_Hand := FALSE;
   Zulauf_AS.BEF_NHV.Bef.BA_Auto := FALSE;
   Zulauf_AS.BEF_NHV.Bef.BF_Ein1 := FALSE;
   Zulauf_AS.BEF_NHV.Bef.BF_Ein2 := FALSE;
   Zulauf_AS.BEF_NHV.Bef.BF_Aus := FALSE;
   Zulauf_AS.BEF_NHV.Bef.BZ_Res := FALSE;
   Zulauf_AS.BEF_NHV.Bef.Res_10 := FALSE;
   Zulauf_AS.BEF_NHV.Bef.Res_11 := FALSE;
   Zulauf_AS.BEF_NHV.Bef.Res_12 := FALSE;
   Zulauf_AS.BEF_NHV.Bef.Res_13 := FALSE;
   Zulauf_AS.BEF_NHV.Bef.Res_14 := FALSE;
   Zulauf_AS.BEF_NHV.Bef.Res_15 := FALSE;
   Zulauf_AS.BEF_NHV.Bef.Res_16 := FALSE;
   Zulauf_AS.BEF_NHV.Bef.Res_17 := FALSE;
   Zulauf_AS.BEF_NHV.Bef.Res_18 := FALSE;
   Zulauf_AS.BEF_NHV.Bef.Res_19 := FALSE;
   Zulauf_AS.BEF_NHV.Bef.Res_20 := FALSE;
   Zulauf_AS.BEF_NHV.Bef.Res_21 := FALSE;
   Zulauf_AS.BEF_NHV.Bef.Res_22 := FALSE;
   Zulauf_AS.BEF_NHV.Bef.Res_23 := FALSE;
   Zulauf_AS.BEF_NHV.Bef.Res_24 := FALSE;
   Zulauf_AS.BEF_NHV.Bef.Res_25 := FALSE;
   Zulauf_AS.BEF_NHV.Bef.Res_26 := FALSE;
   Zulauf_AS.BEF_NHV.Bef.Res_27 := FALSE;
   Zulauf_AS.BEF_NHV.Bef.Res_28 := FALSE;
   Zulauf_AS.BEF_NHV.Bef.Res_29 := FALSE;
   Zulauf_AS.BEF_NHV.Bef.BF_Set_SW_chg := FALSE;
   Zulauf_AS.BEF_NHV.Bef.BF_Quit := FALSE;
   Zulauf_AS.BEF_NHV.SW_Hand := 0.0;
   Zulauf_RA_SA.Typ := 0;
   Zulauf_RA_SA.Idx := 27;
   Zulauf_RA_SA.BA_VW_Hand := FALSE;
   Zulauf_RA_SA.Tmr_VZ_Anlauf_Q := FALSE;
   Zulauf_RA_SA.SS := FALSE;
   Zulauf_RA_SA.SSnq := FALSE;
   Zulauf_RA_SA.SSfq := TRUE;
   Zulauf_RA_SA.nBB := FALSE;
   Zulauf_RA_SA.VW_Hand_St1 := FALSE;
   Zulauf_RA_SA.VW_Hand_St2 := FALSE;
   Zulauf_RA_SA.VW_Hand_Stop := FALSE;
   Zulauf_RA_SA.VW_Auto_St1 := FALSE;
   Zulauf_RA_SA.VW_Auto_St2 := FALSE;
   Zulauf_RA_SA.Anst_Req_St1 := FALSE;
   Zulauf_RA_SA.Anst_Req_St2 := FALSE;
   Zulauf_RA_SA.FM_Betrieb_Ein := FALSE;
   Zulauf_RA_SA.FM_Betrieb_Aus := TRUE;
   Zulauf_RA_SA.NLZ_MAZ_St1 := FALSE;
   Zulauf_RA_SA.NLZ_MAZ_St2 := FALSE;
   Zulauf_RA_SA.NLZ_Rev_SS_St1 := FALSE;
   Zulauf_RA_SA.NLZ_Rev_SS_St2 := FALSE;
   Zulauf_RA_SA.Th_St := FALSE;
   Zulauf_RA_SA.DMA_St := FALSE;
   Zulauf_RA_SA.DMZ_St := FALSE;
   Zulauf_RA_SA.FU_St := FALSE;
   Zulauf_RA_SA.TL_St := FALSE;
   Zulauf_RA_SA.UDr_St := FALSE;
   Zulauf_RA_SA.UeDr_St := FALSE;
   Zulauf_RA_SA.UT_St := FALSE;
   Zulauf_RA_SA.Le_St := FALSE;
   Zulauf_RA_SA.UeLM_St := FALSE;
   Zulauf_RA_SA.UeLE_St := FALSE;
   Zulauf_RA_SA.Kom_DP_St := FALSE;
   Zulauf_RA_SA.Kom_int_St := FALSE;
   Zulauf_RA_SA.int_St := FALSE;
   Zulauf_RA_SA.LZ_St := FALSE;
   Zulauf_RA_SA.BefLZ_St := FALSE;
   Zulauf_RA_SA.FM_GlobalQuit := FALSE;
   Zulauf_RA_SA.Quit_RST := FALSE;
   Zulauf_RA_SA.Tmr_VZ_Anlauf := 0;
   Zulauf_RA_SA.Tmr_VZ_ESZ := 0;
   Zulauf_RA_SA.Tmr_Th_St := 0;
   Zulauf_RA_SA.Tmr_DMA_St := 0;
   Zulauf_RA_SA.Tmr_DMZ_St := 0;
   Zulauf_RA_SA.Tmr_FU_St := 0;
   Zulauf_RA_SA.Tmr_TL_St := 0;
   Zulauf_RA_SA.Tmr_UDr_St := 0;
   Zulauf_RA_SA.Tmr_UeDr_St := 0;
   Zulauf_RA_SA.Tmr_UT_St := 0;
   Zulauf_RA_SA.Tmr_Le_St := 0;
   Zulauf_RA_SA.Tmr_UeLM_St := 0;
   Zulauf_RA_SA.Tmr_UeLE_St := 0;
   Zulauf_RA_SA.Tmr_Kom_DP_St := 0;
   Zulauf_RA_SA.Tmr_Kom_int_St := 0;
   Zulauf_RA_SA.Tmr_int_St := 0;
   Zulauf_RA_SA.Tmr_LZ_St := 0;
   Zulauf_RA_SA.Tmr_BefLZ_St := 0;
   Zulauf_RA_SA.Tmr_ASZ_St1 := 0;
   Zulauf_RA_SA.Tmr_ASZ_St2 := 0;
   Zulauf_RA_SA.Tmr_Rev_St1 := 0;
   Zulauf_RA_SA.Tmr_Rev_St2 := 0;
   Zulauf_RA_SA.BZ_ges_s := 723;
   Zulauf_RA_SA.Tmr_Quit_RST := 0;
   Zulauf_RA_SA.BEF_NHV.Bef.Bed_Res := FALSE;
   Zulauf_RA_SA.BEF_NHV.Bef.Bed_UV := FALSE;
   Zulauf_RA_SA.BEF_NHV.Bef.Bed_NHV := FALSE;
   Zulauf_RA_SA.BEF_NHV.Bef.Bed_PLS := FALSE;
   Zulauf_RA_SA.BEF_NHV.Bef.BA_Hand := FALSE;
   Zulauf_RA_SA.BEF_NHV.Bef.BA_Auto := FALSE;
   Zulauf_RA_SA.BEF_NHV.Bef.BF_Ein1 := FALSE;
   Zulauf_RA_SA.BEF_NHV.Bef.BF_Ein2 := FALSE;
   Zulauf_RA_SA.BEF_NHV.Bef.BF_Aus := FALSE;
   Zulauf_RA_SA.BEF_NHV.Bef.BZ_Res := FALSE;
   Zulauf_RA_SA.BEF_NHV.Bef.Res_10 := FALSE;
   Zulauf_RA_SA.BEF_NHV.Bef.Res_11 := FALSE;
   Zulauf_RA_SA.BEF_NHV.Bef.Res_12 := FALSE;
   Zulauf_RA_SA.BEF_NHV.Bef.Res_13 := FALSE;
   Zulauf_RA_SA.BEF_NHV.Bef.Res_14 := FALSE;
   Zulauf_RA_SA.BEF_NHV.Bef.Res_15 := FALSE;
   Zulauf_RA_SA.BEF_NHV.Bef.Res_16 := FALSE;
   Zulauf_RA_SA.BEF_NHV.Bef.Res_17 := FALSE;
   Zulauf_RA_SA.BEF_NHV.Bef.Res_18 := FALSE;
   Zulauf_RA_SA.BEF_NHV.Bef.Res_19 := FALSE;
   Zulauf_RA_SA.BEF_NHV.Bef.Res_20 := FALSE;
   Zulauf_RA_SA.BEF_NHV.Bef.Res_21 := FALSE;
   Zulauf_RA_SA.BEF_NHV.Bef.Res_22 := FALSE;
   Zulauf_RA_SA.BEF_NHV.Bef.Res_23 := FALSE;
   Zulauf_RA_SA.BEF_NHV.Bef.Res_24 := FALSE;
   Zulauf_RA_SA.BEF_NHV.Bef.Res_25 := FALSE;
   Zulauf_RA_SA.BEF_NHV.Bef.Res_26 := FALSE;
   Zulauf_RA_SA.BEF_NHV.Bef.Res_27 := FALSE;
   Zulauf_RA_SA.BEF_NHV.Bef.Res_28 := FALSE;
   Zulauf_RA_SA.BEF_NHV.Bef.Res_29 := FALSE;
   Zulauf_RA_SA.BEF_NHV.Bef.BF_Set_SW_chg := FALSE;
   Zulauf_RA_SA.BEF_NHV.Bef.BF_Quit := FALSE;
   Zulauf_RA_SA.BEF_NHV.SW_Hand := 0.0;
   Zulauf_RA_HZS.Typ := 0;
   Zulauf_RA_HZS.Idx := 28;
   Zulauf_RA_HZS.BA_VW_Hand := FALSE;
   Zulauf_RA_HZS.Tmr_VZ_Anlauf_Q := FALSE;
   Zulauf_RA_HZS.SS := FALSE;
   Zulauf_RA_HZS.SSnq := FALSE;
   Zulauf_RA_HZS.SSfq := TRUE;
   Zulauf_RA_HZS.nBB := FALSE;
   Zulauf_RA_HZS.VW_Hand_St1 := FALSE;
   Zulauf_RA_HZS.VW_Hand_St2 := FALSE;
   Zulauf_RA_HZS.VW_Hand_Stop := FALSE;
   Zulauf_RA_HZS.VW_Auto_St1 := FALSE;
   Zulauf_RA_HZS.VW_Auto_St2 := FALSE;
   Zulauf_RA_HZS.Anst_Req_St1 := FALSE;
   Zulauf_RA_HZS.Anst_Req_St2 := FALSE;
   Zulauf_RA_HZS.FM_Betrieb_Ein := FALSE;
   Zulauf_RA_HZS.FM_Betrieb_Aus := TRUE;
   Zulauf_RA_HZS.NLZ_MAZ_St1 := FALSE;
   Zulauf_RA_HZS.NLZ_MAZ_St2 := FALSE;
   Zulauf_RA_HZS.NLZ_Rev_SS_St1 := FALSE;
   Zulauf_RA_HZS.NLZ_Rev_SS_St2 := FALSE;
   Zulauf_RA_HZS.Th_St := FALSE;
   Zulauf_RA_HZS.DMA_St := FALSE;
   Zulauf_RA_HZS.DMZ_St := FALSE;
   Zulauf_RA_HZS.FU_St := FALSE;
   Zulauf_RA_HZS.TL_St := FALSE;
   Zulauf_RA_HZS.UDr_St := FALSE;
   Zulauf_RA_HZS.UeDr_St := FALSE;
   Zulauf_RA_HZS.UT_St := FALSE;
   Zulauf_RA_HZS.Le_St := FALSE;
   Zulauf_RA_HZS.UeLM_St := FALSE;
   Zulauf_RA_HZS.UeLE_St := FALSE;
   Zulauf_RA_HZS.Kom_DP_St := FALSE;
   Zulauf_RA_HZS.Kom_int_St := FALSE;
   Zulauf_RA_HZS.int_St := FALSE;
   Zulauf_RA_HZS.LZ_St := FALSE;
   Zulauf_RA_HZS.BefLZ_St := FALSE;
   Zulauf_RA_HZS.FM_GlobalQuit := FALSE;
   Zulauf_RA_HZS.Quit_RST := FALSE;
   Zulauf_RA_HZS.Tmr_VZ_Anlauf := 0;
   Zulauf_RA_HZS.Tmr_VZ_ESZ := 0;
   Zulauf_RA_HZS.Tmr_Th_St := 0;
   Zulauf_RA_HZS.Tmr_DMA_St := 0;
   Zulauf_RA_HZS.Tmr_DMZ_St := 0;
   Zulauf_RA_HZS.Tmr_FU_St := 0;
   Zulauf_RA_HZS.Tmr_TL_St := 0;
   Zulauf_RA_HZS.Tmr_UDr_St := 0;
   Zulauf_RA_HZS.Tmr_UeDr_St := 0;
   Zulauf_RA_HZS.Tmr_UT_St := 0;
   Zulauf_RA_HZS.Tmr_Le_St := 0;
   Zulauf_RA_HZS.Tmr_UeLM_St := 0;
   Zulauf_RA_HZS.Tmr_UeLE_St := 0;
   Zulauf_RA_HZS.Tmr_Kom_DP_St := 0;
   Zulauf_RA_HZS.Tmr_Kom_int_St := 0;
   Zulauf_RA_HZS.Tmr_int_St := 0;
   Zulauf_RA_HZS.Tmr_LZ_St := 0;
   Zulauf_RA_HZS.Tmr_BefLZ_St := 0;
   Zulauf_RA_HZS.Tmr_ASZ_St1 := 0;
   Zulauf_RA_HZS.Tmr_ASZ_St2 := 0;
   Zulauf_RA_HZS.Tmr_Rev_St1 := 0;
   Zulauf_RA_HZS.Tmr_Rev_St2 := 0;
   Zulauf_RA_HZS.BZ_ges_s := 2227;
   Zulauf_RA_HZS.Tmr_Quit_RST := 0;
   Zulauf_RA_HZS.BEF_NHV.Bef.Bed_Res := FALSE;
   Zulauf_RA_HZS.BEF_NHV.Bef.Bed_UV := FALSE;
   Zulauf_RA_HZS.BEF_NHV.Bef.Bed_NHV := FALSE;
   Zulauf_RA_HZS.BEF_NHV.Bef.Bed_PLS := FALSE;
   Zulauf_RA_HZS.BEF_NHV.Bef.BA_Hand := FALSE;
   Zulauf_RA_HZS.BEF_NHV.Bef.BA_Auto := FALSE;
   Zulauf_RA_HZS.BEF_NHV.Bef.BF_Ein1 := FALSE;
   Zulauf_RA_HZS.BEF_NHV.Bef.BF_Ein2 := FALSE;
   Zulauf_RA_HZS.BEF_NHV.Bef.BF_Aus := FALSE;
   Zulauf_RA_HZS.BEF_NHV.Bef.BZ_Res := FALSE;
   Zulauf_RA_HZS.BEF_NHV.Bef.Res_10 := FALSE;
   Zulauf_RA_HZS.BEF_NHV.Bef.Res_11 := FALSE;
   Zulauf_RA_HZS.BEF_NHV.Bef.Res_12 := FALSE;
   Zulauf_RA_HZS.BEF_NHV.Bef.Res_13 := FALSE;
   Zulauf_RA_HZS.BEF_NHV.Bef.Res_14 := FALSE;
   Zulauf_RA_HZS.BEF_NHV.Bef.Res_15 := FALSE;
   Zulauf_RA_HZS.BEF_NHV.Bef.Res_16 := FALSE;
   Zulauf_RA_HZS.BEF_NHV.Bef.Res_17 := FALSE;
   Zulauf_RA_HZS.BEF_NHV.Bef.Res_18 := FALSE;
   Zulauf_RA_HZS.BEF_NHV.Bef.Res_19 := FALSE;
   Zulauf_RA_HZS.BEF_NHV.Bef.Res_20 := FALSE;
   Zulauf_RA_HZS.BEF_NHV.Bef.Res_21 := FALSE;
   Zulauf_RA_HZS.BEF_NHV.Bef.Res_22 := FALSE;
   Zulauf_RA_HZS.BEF_NHV.Bef.Res_23 := FALSE;
   Zulauf_RA_HZS.BEF_NHV.Bef.Res_24 := FALSE;
   Zulauf_RA_HZS.BEF_NHV.Bef.Res_25 := FALSE;
   Zulauf_RA_HZS.BEF_NHV.Bef.Res_26 := FALSE;
   Zulauf_RA_HZS.BEF_NHV.Bef.Res_27 := FALSE;
   Zulauf_RA_HZS.BEF_NHV.Bef.Res_28 := FALSE;
   Zulauf_RA_HZS.BEF_NHV.Bef.Res_29 := FALSE;
   Zulauf_RA_HZS.BEF_NHV.Bef.BF_Set_SW_chg := FALSE;
   Zulauf_RA_HZS.BEF_NHV.Bef.BF_Quit := FALSE;
   Zulauf_RA_HZS.BEF_NHV.SW_Hand := 0.0;
   Zulauf_RA_VKS.Typ := 0;
   Zulauf_RA_VKS.Idx := 29;
   Zulauf_RA_VKS.BA_VW_Hand := FALSE;
   Zulauf_RA_VKS.Tmr_VZ_Anlauf_Q := FALSE;
   Zulauf_RA_VKS.SS := FALSE;
   Zulauf_RA_VKS.SSnq := FALSE;
   Zulauf_RA_VKS.SSfq := TRUE;
   Zulauf_RA_VKS.nBB := FALSE;
   Zulauf_RA_VKS.VW_Hand_St1 := FALSE;
   Zulauf_RA_VKS.VW_Hand_St2 := FALSE;
   Zulauf_RA_VKS.VW_Hand_Stop := FALSE;
   Zulauf_RA_VKS.VW_Auto_St1 := FALSE;
   Zulauf_RA_VKS.VW_Auto_St2 := FALSE;
   Zulauf_RA_VKS.Anst_Req_St1 := FALSE;
   Zulauf_RA_VKS.Anst_Req_St2 := FALSE;
   Zulauf_RA_VKS.FM_Betrieb_Ein := FALSE;
   Zulauf_RA_VKS.FM_Betrieb_Aus := TRUE;
   Zulauf_RA_VKS.NLZ_MAZ_St1 := FALSE;
   Zulauf_RA_VKS.NLZ_MAZ_St2 := FALSE;
   Zulauf_RA_VKS.NLZ_Rev_SS_St1 := FALSE;
   Zulauf_RA_VKS.NLZ_Rev_SS_St2 := FALSE;
   Zulauf_RA_VKS.Th_St := FALSE;
   Zulauf_RA_VKS.DMA_St := FALSE;
   Zulauf_RA_VKS.DMZ_St := FALSE;
   Zulauf_RA_VKS.FU_St := FALSE;
   Zulauf_RA_VKS.TL_St := FALSE;
   Zulauf_RA_VKS.UDr_St := FALSE;
   Zulauf_RA_VKS.UeDr_St := FALSE;
   Zulauf_RA_VKS.UT_St := FALSE;
   Zulauf_RA_VKS.Le_St := FALSE;
   Zulauf_RA_VKS.UeLM_St := FALSE;
   Zulauf_RA_VKS.UeLE_St := FALSE;
   Zulauf_RA_VKS.Kom_DP_St := FALSE;
   Zulauf_RA_VKS.Kom_int_St := FALSE;
   Zulauf_RA_VKS.int_St := FALSE;
   Zulauf_RA_VKS.LZ_St := FALSE;
   Zulauf_RA_VKS.BefLZ_St := FALSE;
   Zulauf_RA_VKS.FM_GlobalQuit := FALSE;
   Zulauf_RA_VKS.Quit_RST := FALSE;
   Zulauf_RA_VKS.Tmr_VZ_Anlauf := 0;
   Zulauf_RA_VKS.Tmr_VZ_ESZ := 0;
   Zulauf_RA_VKS.Tmr_Th_St := 0;
   Zulauf_RA_VKS.Tmr_DMA_St := 0;
   Zulauf_RA_VKS.Tmr_DMZ_St := 0;
   Zulauf_RA_VKS.Tmr_FU_St := 0;
   Zulauf_RA_VKS.Tmr_TL_St := 0;
   Zulauf_RA_VKS.Tmr_UDr_St := 0;
   Zulauf_RA_VKS.Tmr_UeDr_St := 0;
   Zulauf_RA_VKS.Tmr_UT_St := 0;
   Zulauf_RA_VKS.Tmr_Le_St := 0;
   Zulauf_RA_VKS.Tmr_UeLM_St := 0;
   Zulauf_RA_VKS.Tmr_UeLE_St := 0;
   Zulauf_RA_VKS.Tmr_Kom_DP_St := 0;
   Zulauf_RA_VKS.Tmr_Kom_int_St := 0;
   Zulauf_RA_VKS.Tmr_int_St := 0;
   Zulauf_RA_VKS.Tmr_LZ_St := 0;
   Zulauf_RA_VKS.Tmr_BefLZ_St := 0;
   Zulauf_RA_VKS.Tmr_ASZ_St1 := 0;
   Zulauf_RA_VKS.Tmr_ASZ_St2 := 0;
   Zulauf_RA_VKS.Tmr_Rev_St1 := 0;
   Zulauf_RA_VKS.Tmr_Rev_St2 := 0;
   Zulauf_RA_VKS.BZ_ges_s := 1059;
   Zulauf_RA_VKS.Tmr_Quit_RST := 0;
   Zulauf_RA_VKS.BEF_NHV.Bef.Bed_Res := FALSE;
   Zulauf_RA_VKS.BEF_NHV.Bef.Bed_UV := FALSE;
   Zulauf_RA_VKS.BEF_NHV.Bef.Bed_NHV := FALSE;
   Zulauf_RA_VKS.BEF_NHV.Bef.Bed_PLS := FALSE;
   Zulauf_RA_VKS.BEF_NHV.Bef.BA_Hand := FALSE;
   Zulauf_RA_VKS.BEF_NHV.Bef.BA_Auto := FALSE;
   Zulauf_RA_VKS.BEF_NHV.Bef.BF_Ein1 := FALSE;
   Zulauf_RA_VKS.BEF_NHV.Bef.BF_Ein2 := FALSE;
   Zulauf_RA_VKS.BEF_NHV.Bef.BF_Aus := FALSE;
   Zulauf_RA_VKS.BEF_NHV.Bef.BZ_Res := FALSE;
   Zulauf_RA_VKS.BEF_NHV.Bef.Res_10 := FALSE;
   Zulauf_RA_VKS.BEF_NHV.Bef.Res_11 := FALSE;
   Zulauf_RA_VKS.BEF_NHV.Bef.Res_12 := FALSE;
   Zulauf_RA_VKS.BEF_NHV.Bef.Res_13 := FALSE;
   Zulauf_RA_VKS.BEF_NHV.Bef.Res_14 := FALSE;
   Zulauf_RA_VKS.BEF_NHV.Bef.Res_15 := FALSE;
   Zulauf_RA_VKS.BEF_NHV.Bef.Res_16 := FALSE;
   Zulauf_RA_VKS.BEF_NHV.Bef.Res_17 := FALSE;
   Zulauf_RA_VKS.BEF_NHV.Bef.Res_18 := FALSE;
   Zulauf_RA_VKS.BEF_NHV.Bef.Res_19 := FALSE;
   Zulauf_RA_VKS.BEF_NHV.Bef.Res_20 := FALSE;
   Zulauf_RA_VKS.BEF_NHV.Bef.Res_21 := FALSE;
   Zulauf_RA_VKS.BEF_NHV.Bef.Res_22 := FALSE;
   Zulauf_RA_VKS.BEF_NHV.Bef.Res_23 := FALSE;
   Zulauf_RA_VKS.BEF_NHV.Bef.Res_24 := FALSE;
   Zulauf_RA_VKS.BEF_NHV.Bef.Res_25 := FALSE;
   Zulauf_RA_VKS.BEF_NHV.Bef.Res_26 := FALSE;
   Zulauf_RA_VKS.BEF_NHV.Bef.Res_27 := FALSE;
   Zulauf_RA_VKS.BEF_NHV.Bef.Res_28 := FALSE;
   Zulauf_RA_VKS.BEF_NHV.Bef.Res_29 := FALSE;
   Zulauf_RA_VKS.BEF_NHV.Bef.BF_Set_SW_chg := FALSE;
   Zulauf_RA_VKS.BEF_NHV.Bef.BF_Quit := FALSE;
   Zulauf_RA_VKS.BEF_NHV.SW_Hand := 0.0;
   Zulauf_RA_V.Typ := 0;
   Zulauf_RA_V.Idx := 30;
   Zulauf_RA_V.BA_VW_Hand := FALSE;
